C05458=1092.855,441.549,394.876,178.684,26.061,154.074
C05459=1092.862,441.795,394.832,178.687,26.074,154.077
C05460=1092.868,442.041,394.788,178.690,26.088,154.080
C05461=1092.875,442.287,394.744,178.693,26.101,154.083
C05462=1092.881,442.532,394.701,178.697,26.115,154.086
C05463=1092.888,442.778,394.656,178.700,26.128,154.089
C05464=1092.894,443.024,394.612,178.703,26.142,154.092
C05465=1092.901,443.270,394.568,178.707,26.155,154.095
C05466=1092.908,443.516,394.523,178.710,26.169,154.098
C05467=1092.914,443.762,394.479,178.713,26.182,154.101
C05468=1092.921,444.007,394.435,178.716,26.196,154.104
C05469=1092.927,444.253,394.390,178.719,26.210,154.107
C05470=1092.934,444.499,394.346,178.723,26.224,154.110
C05471=1092.941,444.745,394.302,178.725,26.237,154.114
C05472=1092.947,444.991,394.257,178.728,26.251,154.117
C05473=1092.954,445.237,394.213,178.730,26.265,154.120
C05474=1092.960,445.482,394.169,178.733,26.279,154.123
C05475=1092.968,445.728,394.124,178.735,26.292,154.126
C05476=1092.973,445.974,394.079,178.737,26.306,154.130
C05477=1092.980,446.220,394.035,178.738,26.319,154.133
C05478=1092.988,446.466,393.990,178.741,26.333,154.136
C05479=1092.994,446.712,393.946,178.741,26.347,154.140
C05480=1093.000,446.958,393.901,178.743,26.361,154.143
C05481=1093.007,447.204,393.856,178.744,26.374,154.146
C05482=1093.014,447.449,393.811,178.745,26.388,154.150
C05483=1093.020,447.695,393.767,178.746,26.401,154.153
C05484=1093.027,447.941,393.722,178.747,26.415,154.156
C05485=1093.034,448.187,393.677,178.747,26.429,154.160
C05486=1093.040,448.432,393.632,178.747,26.442,154.163
C05487=1093.047,448.678,393.587,178.748,26.456,154.166
C05488=1093.054,448.924,393.543,178.748,26.469,154.170
C05489=1093.060,449.170,393.497,178.748,26.483,154.173
C05490=1093.067,449.415,393.453,178.747,26.496,154.177
C05491=1093.074,449.661,393.408,178.748,26.510,154.180
C05492=1093.081,449.906,393.363,178.748,26.523,154.184
C05493=1093.089,450.153,393.319,178.747,26.535,154.187
C05494=1092.703,450.144,393.142,178.697,26.740,154.244
C05495=1092.694,449.897,393.187,178.697,26.727,154.241
C05496=1092.687,449.651,393.232,178.698,26.714,154.237
C05497=1092.680,449.406,393.276,178.698,26.700,154.234
C05498=1092.673,449.161,393.321,178.698,26.686,154.230
C05499=1092.667,448.915,393.366,178.698,26.673,154.227
C05500=1092.660,448.669,393.411,178.698,26.660,154.224
C05501=1092.653,448.423,393.456,178.697,26.646,154.220
C05502=1092.647,448.177,393.501,178.697,26.633,154.217
C05503=1092.640,447.932,393.546,178.697,26.619,154.213
C05504=1092.633,447.686,393.591,178.695,26.605,154.210
C05505=1092.627,447.440,393.636,178.695,26.591,154.207
C05506=1092.620,447.195,393.680,178.694,26.578,154.203
C05507=1092.613,446.949,393.725,178.692,26.564,154.200
C05508=1092.607,446.702,393.770,178.691,26.550,154.197
C05509=1092.600,446.457,393.814,178.689,26.536,154.193
C05510=1092.593,446.211,393.859,178.687,26.523,154.190
C05511=1092.586,445.966,393.904,178.686,26.509,154.187
C05512=1092.580,445.719,393.948,178.684,26.495,154.183
C05513=1092.573,445.473,393.993,178.682,26.482,154.180
C05514=1092.566,445.228,394.038,178.679,26.468,154.177
C05515=1092.560,444.982,394.082,178.677,26.454,154.174
C05516=1092.553,444.736,394.126,178.674,26.440,154.170
C05517=1092.547,444.490,394.172,178.671,26.427,154.167
C05518=1092.540,444.244,394.215,178.668,26.413,154.164
C05519=1092.533,443.999,394.260,178.664,26.399,154.161
C05520=1092.526,443.752,394.304,178.661,26.385,154.158
C05521=1092.520,443.507,394.349,178.658,26.371,154.155
C05522=1092.513,443.261,394.393,178.655,26.358,154.152
C05523=1092.507,443.016,394.437,178.651,26.344,154.149
C05524=1092.500,442.770,394.481,178.647,26.330,154.146
C05525=1092.493,442.524,394.526,178.644,26.317,154.143
C05526=1092.487,442.278,394.569,178.641,26.303,154.139
C05527=1092.480,442.032,394.614,178.638,26.290,154.136
C05528=1092.474,441.786,394.658,178.634,26.276,154.133
C05529=1092.467,441.540,394.702,178.631,26.263,154.130
C05530=1092.460,441.294,394.746,178.628,26.250,154.127
C05531=1092.454,441.048,394.790,178.624,26.237,154.125
C05532=1092.448,440.802,394.834,178.621,26.224,154.122
C05533=1092.441,440.556,394.878,178.618,26.210,154.119
C05534=1092.434,440.311,394.922,178.614,26.197,154.116
C05535=1092.428,440.065,394.966,178.611,26.185,154.113
C05536=1092.421,439.818,395.010,178.608,26.171,154.110
C05537=1092.414,439.573,395.053,178.604,26.158,154.107
C05538=1092.407,439.327,395.097,178.601,26.146,154.104
C05539=1092.397,438.921,395.169,178.596,26.124,154.099
C05540=1092.386,438.515,395.241,178.590,26.104,154.095
C05541=1092.375,438.111,395.313,178.585,26.083,154.090
C05542=1092.364,437.705,395.384,178.579,26.062,154.086
C05543=1092.358,437.459,395.428,178.576,26.050,154.083
C05544=1092.351,437.214,395.471,178.573,26.037,154.080
C05545=1092.345,436.967,395.514,178.570,26.025,154.077
C05546=1092.338,436.721,395.558,178.566,26.012,154.075
C05547=1092.331,436.475,395.602,178.562,25.999,154.072
C05548=1092.325,436.229,395.645,178.560,25.987,154.069
C05549=1092.319,435.983,395.689,178.556,25.975,154.066
C05550=1092.311,435.737,395.732,178.553,25.963,154.064
C05551=1092.306,435.491,395.775,178.550,25.951,154.061
C05552=1092.300,435.245,395.818,178.546,25.938,154.058
C05553=1092.293,434.999,395.861,178.544,25.927,154.056
C05554=1092.286,434.753,395.905,178.540,25.914,154.053
C05555=1092.279,434.507,395.947,178.537,25.902,154.050
C05556=1092.273,434.260,395.990,178.533,25.890,154.048
C05557=1092.267,434.015,396.034,178.530,25.878,154.045
C05558=1092.261,433.769,396.076,178.527,25.866,154.042
C05559=1092.254,433.522,396.120,178.524,25.854,154.040
C05560=1092.247,433.276,396.163,178.521,25.843,154.037
C05561=1092.242,433.030,396.206,178.517,25.831,154.035
C05562=1092.235,432.784,396.248,178.514,25.819,154.032
C05563=1092.229,432.538,396.291,178.510,25.807,154.029
C05564=1092.222,432.291,396.334,178.508,25.796,154.027
C05565=1092.215,432.046,396.377,178.505,25.784,154.024
C05566=1092.209,431.800,396.420,178.501,25.772,154.022
C05567=1092.202,431.553,396.462,178.498,25.761,154.019
C05568=1092.196,431.307,396.506,178.495,25.750,154.017
C05569=1092.189,431.061,396.548,178.491,25.738,154.014
C05570=1092.183,430.815,396.590,178.488,25.726,154.012
C05571=1092.177,430.568,396.633,178.485,25.716,154.010
C05572=1092.170,430.322,396.676,178.481,25.704,154.007
C05573=1092.164,430.077,396.718,178.478,25.692,154.005
C05574=1092.158,429.830,396.761,178.475,25.681,154.002
C05575=1092.151,429.584,396.804,178.472,25.670,154.000
C05576=1092.145,429.337,396.845,178.469,25.659,153.997
C05577=1092.138,429.091,396.888,178.466,25.648,153.995
C05578=1092.132,428.845,396.931,178.463,25.637,153.993
C05579=1092.126,428.599,396.973,178.459,25.625,153.990
C05580=1092.119,428.352,397.015,178.456,25.614,153.988
C05581=1092.112,428.106,397.057,178.453,25.603,153.985
C05582=1092.106,427.860,397.100,178.449,25.593,153.983
C05583=1092.100,427.613,397.141,178.447,25.582,153.981
C05584=1092.093,427.367,397.185,178.443,25.571,153.978
C05585=1092.087,427.121,397.227,178.440,25.560,153.976
C05586=1092.081,426.874,397.269,178.437,25.549,153.974
C05587=1092.074,426.629,397.311,178.433,25.539,153.972
C05588=1092.068,426.382,397.353,178.430,25.528,153.969
C05589=1092.062,426.136,397.395,178.427,25.518,153.967
C05590=1092.055,425.889,397.437,178.423,25.507,153.965
C05591=1092.049,425.658,397.476,178.421,25.497,153.963
C05592=1092.043,425.427,397.515,178.418,25.487,153.961
C05593=1092.037,425.196,397.555,178.415,25.477,153.958
C05594=1092.031,424.965,397.594,178.411,25.467,153.956
C05595=1092.025,424.733,397.634,178.409,25.457,153.954
C05596=1092.019,424.503,397.673,178.406,25.447,153.952
C05597=1092.013,424.271,397.713,178.403,25.437,153.950
C05598=1092.008,424.040,397.751,178.399,25.427,153.948
C05599=1092.001,423.793,397.794,178.396,25.417,153.946
C05600=1091.995,423.547,397.835,178.393,25.407,153.944
C05601=1091.988,423.300,397.877,178.390,25.396,153.941
C05602=1091.982,423.054,397.918,178.387,25.386,153.939
C05603=1091.976,422.807,397.960,178.384,25.376,153.937
C05604=1091.970,422.562,398.002,178.381,25.366,153.935
C05605=1091.963,422.315,398.044,178.377,25.356,153.933
C05606=1091.957,422.069,398.086,178.374,25.345,153.931
C05607=1091.951,421.822,398.127,178.371,25.335,153.929
C05608=1091.944,421.576,398.168,178.368,25.325,153.926
C05609=1091.938,421.330,398.210,178.365,25.316,153.924
C05610=1091.931,421.083,398.252,178.362,25.305,153.922
C05611=1091.925,420.836,398.293,178.358,25.295,153.920
C05612=1091.919,420.591,398.334,178.355,25.286,153.918
C05613=1091.913,420.343,398.375,178.352,25.275,153.916
C05614=1091.907,420.097,398.416,178.349,25.266,153.914
C05615=1091.900,419.850,398.458,178.345,25.256,153.912
C05616=1091.893,419.604,398.499,178.342,25.246,153.910
C05617=1091.887,419.358,398.541,178.339,25.236,153.908
C05618=1091.881,419.111,398.582,178.336,25.227,153.906
C05619=1091.874,418.864,398.623,178.334,25.217,153.904
C05620=1091.869,418.618,398.664,178.330,25.208,153.902
C05621=1091.863,418.372,398.705,178.327,25.198,153.900
C05622=1091.856,418.124,398.747,178.324,25.188,153.898
C05623=1091.850,417.879,398.787,178.321,25.179,153.896
C05624=1091.844,417.632,398.829,178.317,25.169,153.894
C05625=1091.838,417.386,398.870,178.314,25.159,153.892
C05626=1091.831,417.139,398.911,178.311,25.150,153.890
C05627=1091.821,416.758,398.974,178.306,25.135,153.887
C05628=1091.812,416.375,399.038,178.301,25.120,153.884
C05629=1091.803,415.993,399.101,178.296,25.106,153.881
C05630=1091.793,415.612,399.165,178.292,25.092,153.878
C05631=1091.786,415.365,399.205,178.288,25.082,153.876
C05632=1091.780,415.119,399.245,178.286,25.074,153.874
C05633=1091.773,414.872,399.287,178.282,25.064,153.873
C05634=1091.767,414.625,399.327,178.279,25.055,153.871
C05635=1091.761,414.378,399.368,178.276,25.046,153.869
C05636=1091.755,414.133,399.409,178.273,25.037,153.867
C05637=1091.748,413.886,399.449,178.270,25.028,153.865
C05638=1091.742,413.638,399.490,178.267,25.018,153.863
C05639=1091.736,413.392,399.530,178.263,25.010,153.861
C05640=1091.730,413.146,399.571,178.261,25.001,153.860
C05641=1091.723,412.899,399.612,178.258,24.992,153.858
C05642=1091.717,412.653,399.652,178.254,24.983,153.856
C05643=1091.711,412.406,399.692,178.251,24.973,153.854
C05644=1091.705,412.159,399.733,178.248,24.965,153.852
C05645=1091.698,411.913,399.773,178.245,24.956,153.851
C05646=1091.692,411.665,399.814,178.242,24.947,153.849
C05647=1091.685,411.354,399.865,178.238,24.936,153.847
C05648=1091.676,411.041,399.916,178.234,24.925,153.844
C05649=1091.668,410.729,399.967,178.230,24.914,153.842
C05650=1091.661,410.417,400.017,178.226,24.903,153.840
C05651=1091.655,410.170,400.058,178.223,24.894,153.838
C05652=1091.649,409.924,400.098,178.221,24.885,153.836
C05653=1091.642,409.677,400.138,178.217,24.877,153.835
C05654=1091.636,409.431,400.179,178.214,24.868,153.833
C05655=1091.631,409.183,400.219,178.211,24.860,153.831
C05656=1091.624,408.937,400.259,178.208,24.851,153.829
C05657=1091.618,408.690,400.299,178.205,24.842,153.828
C05658=1091.611,408.444,400.339,178.202,24.834,153.826
C05659=1091.606,408.196,400.379,178.198,24.825,153.824
C05660=1091.600,407.950,400.419,178.196,24.817,153.823
C05661=1091.593,407.703,400.459,178.192,24.808,153.821
C05662=1091.587,407.457,400.500,178.190,24.800,153.819
C05663=1091.581,407.210,400.539,178.186,24.791,153.818
C05664=1091.575,406.963,400.579,178.184,24.783,153.816
C05665=1091.568,406.716,400.619,178.180,24.775,153.814
C05666=1091.562,406.469,400.659,178.177,24.767,153.813
C05667=1091.557,406.223,400.699,178.174,24.758,153.811
C05668=1091.551,405.976,400.739,178.171,24.750,153.809
C05669=1091.545,405.730,400.779,178.168,24.742,153.808
C05670=1091.539,405.482,400.818,178.165,24.734,153.806
C05671=1091.532,405.236,400.858,178.162,24.725,153.805
C05672=1091.526,404.989,400.898,178.159,24.718,153.803
C05673=1091.520,404.742,400.937,178.156,24.709,153.801
C05674=1091.514,404.495,400.977,178.153,24.701,153.800
C05675=1091.508,404.249,401.016,178.149,24.693,153.798
C05676=1091.501,404.003,401.056,178.147,24.685,153.797
C05677=1091.495,403.755,401.095,178.143,24.677,153.795
C05678=1091.489,403.508,401.135,178.141,24.669,153.794
C05679=1091.483,403.261,401.174,178.138,24.661,153.792
C05680=1091.476,403.015,401.214,178.134,24.653,153.791
C05681=1091.471,402.768,401.253,178.132,24.645,153.789
C05682=1091.465,402.521,401.293,178.128,24.637,153.787
C05683=1091.458,402.274,401.332,178.125,24.630,153.786
C05684=1091.452,402.028,401.372,178.123,24.622,153.784
C05685=1091.446,401.781,401.411,178.119,24.614,153.783
C05686=1091.440,401.534,401.450,178.116,24.606,153.781
C05687=1091.434,401.287,401.490,178.113,24.598,153.780
C05688=1091.427,401.040,401.529,178.110,24.591,153.778
C05689=1091.422,400.794,401.568,178.107,24.583,153.777
C05690=1091.416,400.547,401.607,178.104,24.575,153.775
C05691=1091.410,400.299,401.647,178.101,24.568,153.774
C05692=1091.403,400.053,401.685,178.098,24.560,153.772
C05693=1091.397,399.806,401.724,178.095,24.552,153.771
C05694=1091.391,399.559,401.764,178.092,24.544,153.769
C05695=1091.385,399.312,401.803,178.089,24.537,153.768
C05696=1091.379,399.066,401.842,178.086,24.529,153.767
C05697=1091.373,398.819,401.881,178.083,24.522,153.765
C05698=1091.367,398.572,401.921,178.080,24.514,153.764
C05699=1091.361,398.349,401.956,178.077,24.508,153.762
C05700=1091.355,398.126,401.991,178.074,24.500,153.761
C05701=1091.351,397.902,402.026,178.071,24.494,153.760
C05702=1091.345,397.679,402.061,178.069,24.487,153.759
C05703=1091.339,397.455,402.097,178.066,24.480,153.757
C05704=1091.333,397.232,402.132,178.063,24.474,153.756
C05705=1091.328,397.008,402.166,178.060,24.467,153.755
C05706=1091.323,396.785,402.202,178.058,24.461,153.753
C05707=1091.316,396.538,402.241,178.055,24.453,153.752
C05708=1091.311,396.291,402.279,178.052,24.446,153.751
C05709=1091.304,396.044,402.318,178.049,24.438,153.749
C05710=1091.299,395.798,402.357,178.046,24.431,153.748
C05711=1091.292,395.551,402.395,178.043,24.424,153.747
C05712=1091.287,395.304,402.434,178.040,24.417,153.745
C05713=1091.280,395.057,402.473,178.037,24.409,153.744
C05714=1091.275,394.810,402.512,178.034,24.402,153.742
C05715=1091.268,394.563,402.550,178.030,24.395,153.741
C05716=1091.262,394.316,402.589,178.028,24.388,153.740
C05717=1091.256,394.070,402.628,178.025,24.380,153.738
C05718=1091.249,393.823,402.666,178.022,24.373,153.737
C05719=1091.244,393.576,402.705,178.019,24.367,153.736
C05720=1091.237,393.328,402.743,178.015,24.359,153.734
C05721=1091.232,393.082,402.782,178.012,24.352,153.733
C05722=1091.226,392.835,402.820,178.009,24.345,153.732
C05723=1091.219,392.588,402.859,178.007,24.338,153.730
C05724=1091.214,392.341,402.897,178.004,24.331,153.729
C05725=1091.207,392.094,402.936,178.001,24.324,153.728
C05726=1091.201,391.848,402.974,177.997,24.317,153.727
C05727=1091.195,391.600,403.012,177.994,24.310,153.725
C05728=1091.189,391.354,403.051,177.991,24.303,153.724
C05729=1091.183,391.106,403.089,177.988,24.296,153.723
C05730=1091.177,390.860,403.127,177.985,24.290,153.722
C05731=1091.171,390.613,403.165,177.982,24.283,153.720
C05732=1091.164,390.366,403.203,177.979,24.275,153.719
C05733=1091.158,390.119,403.241,177.976,24.269,153.718
C05734=1091.152,389.872,403.279,177.973,24.262,153.717
C05735=1091.147,389.625,403.317,177.970,24.255,153.715
C05736=1091.140,389.379,403.356,177.967,24.249,153.714
C05737=1091.134,389.131,403.394,177.964,24.242,153.713
C05738=1091.128,388.884,403.432,177.961,24.235,153.712
C05739=1091.122,388.638,403.470,177.957,24.228,153.710
C05740=1091.116,388.390,403.508,177.954,24.222,153.709
C05741=1091.110,388.143,403.545,177.951,24.215,153.708
C05742=1091.104,387.897,403.583,177.948,24.208,153.707
C05743=1091.098,387.650,403.621,177.945,24.202,153.706
C05744=1091.091,387.403,403.659,177.943,24.195,153.704
C05745=1091.086,387.156,403.697,177.939,24.189,153.703
C05746=1091.080,386.909,403.735,177.937,24.182,153.702
C05747=1091.074,386.662,403.773,177.934,24.175,153.701
C05748=1091.068,386.415,403.811,177.931,24.169,153.700
C05749=1091.062,386.168,403.849,177.927,24.162,153.699
C05750=1091.056,385.921,403.887,177.924,24.156,153.697
C05751=1091.050,385.674,403.924,177.921,24.149,153.696
C05752=1091.044,385.427,403.962,177.918,24.143,153.695
C05753=1091.038,385.180,404.000,177.915,24.136,153.694
C05754=1091.032,384.933,404.038,177.912,24.130,153.693
C05755=1091.026,384.716,404.071,177.910,24.124,153.692
C05756=1091.021,384.500,404.103,177.906,24.118,153.691
C05757=1091.016,384.282,404.137,177.904,24.113,153.690
C05758=1091.011,384.066,404.169,177.901,24.107,153.689
C05759=1091.005,383.849,404.203,177.898,24.101,153.688
C05760=1091.000,383.633,404.236,177.896,24.095,153.687
C05761=1090.995,383.416,404.269,177.893,24.090,153.686
C05762=1090.991,383.199,404.302,177.891,24.084,153.685
C05763=1090.985,382.952,404.339,177.888,24.078,153.684
C05764=1090.978,382.705,404.376,177.885,24.072,153.682
C05765=1090.972,382.458,404.414,177.882,24.065,153.681
C05766=1090.966,382.211,404.452,177.879,24.059,153.680
C05767=1090.960,381.964,404.489,177.875,24.053,153.679
C05768=1090.954,381.717,404.527,177.872,24.047,153.678
C05769=1090.948,381.470,404.563,177.869,24.040,153.677
C05770=1090.942,381.223,404.601,177.866,24.034,153.676
C05771=1090.937,380.976,404.638,177.863,24.028,153.675
C05772=1090.930,380.729,404.675,177.860,24.022,153.674
C05773=1090.924,380.481,404.712,177.857,24.016,153.673
C05774=1090.918,380.234,404.750,177.854,24.010,153.672
C05775=1090.912,379.987,404.787,177.851,24.003,153.671
C05776=1090.906,379.741,404.824,177.848,23.997,153.670
C05777=1090.900,379.493,404.861,177.845,23.991,153.669
C05778=1090.894,379.246,404.898,177.842,23.985,153.667
C05779=1090.888,378.999,404.936,177.839,23.979,153.666
C05780=1090.882,378.752,404.973,177.835,23.973,153.665
C05781=1090.877,378.505,405.010,177.832,23.967,153.664
C05782=1090.870,378.258,405.047,177.829,23.961,153.663
C05783=1090.864,378.011,405.084,177.827,23.955,153.662
C05784=1090.859,377.764,405.121,177.824,23.949,153.661
C05785=1090.852,377.517,405.157,177.821,23.943,153.660
C05786=1090.846,377.270,405.195,177.818,23.937,153.659
C05787=1090.840,377.023,405.231,177.814,23.931,153.658
C05788=1090.835,376.775,405.269,177.811,23.925,153.657
C05789=1090.829,376.528,405.306,177.808,23.919,153.656
C05790=1090.823,376.281,405.342,177.805,23.913,153.655
C05791=1090.817,376.034,405.380,177.802,23.907,153.654
C05792=1090.811,375.787,405.417,177.799,23.901,153.653
C05793=1090.805,375.540,405.453,177.796,23.895,153.652
C05794=1090.799,375.292,405.490,177.793,23.890,153.651
C05795=1090.793,375.045,405.527,177.790,23.884,153.650
C05796=1090.787,374.798,405.564,177.787,23.878,153.649
C05797=1090.781,374.551,405.600,177.784,23.872,153.648
C05798=1090.775,374.304,405.637,177.781,23.866,153.647
C05799=1090.769,374.057,405.674,177.778,23.860,153.646
C05800=1090.763,373.809,405.711,177.774,23.855,153.645
C05801=1090.758,373.563,405.747,177.771,23.849,153.644
C05802=1090.752,373.315,405.784,177.769,23.843,153.643
C05803=1090.746,373.068,405.820,177.766,23.837,153.642
C05804=1090.740,372.821,405.856,177.763,23.832,153.641
C05805=1090.734,372.573,405.893,177.759,23.826,153.641
C05806=1090.728,372.326,405.930,177.756,23.820,153.640
C05807=1090.721,372.079,405.966,177.753,23.814,153.639
C05808=1090.716,371.832,406.003,177.750,23.809,153.638
C05809=1090.710,371.584,406.039,177.747,23.804,153.637
C05810=1090.703,371.337,406.075,177.744,23.798,153.636
C05811=1090.694,370.932,406.135,177.739,23.789,153.634
C05812=1090.684,370.525,406.195,177.734,23.779,153.633
C05813=1090.675,370.119,406.255,177.729,23.770,153.631
C05814=1090.665,369.714,406.314,177.724,23.761,153.630
C05815=1090.659,369.467,406.350,177.721,23.756,153.629
C05816=1090.652,369.220,406.387,177.718,23.750,153.628
C05817=1090.647,368.972,406.423,177.715,23.744,153.627
C05818=1090.641,368.725,406.459,177.712,23.739,153.626
C05819=1090.635,368.478,406.495,177.708,23.734,153.626
C05820=1090.629,368.231,406.531,177.706,23.728,153.625
C05821=1090.624,367.983,406.568,177.703,23.723,153.624
C05822=1090.618,367.736,406.604,177.699,23.717,153.623
C05823=1090.612,367.489,406.639,177.696,23.712,153.622
C05824=1090.605,367.242,406.676,177.693,23.706,153.621
C05825=1090.600,366.994,406.712,177.691,23.701,153.620
C05826=1090.594,366.747,406.748,177.687,23.696,153.619
C05827=1090.588,366.500,406.784,177.684,23.690,153.618
C05828=1090.582,366.252,406.820,177.681,23.684,153.618
C05829=1090.577,366.006,406.856,177.678,23.679,153.617
C05830=1090.571,365.758,406.892,177.675,23.674,153.616
C05831=1090.565,365.510,406.928,177.672,23.669,153.615
C05832=1090.559,365.263,406.964,177.668,23.663,153.614
C05833=1090.553,365.016,407.000,177.666,23.658,153.613
C05834=1090.547,364.768,407.035,177.663,23.653,153.613
C05835=1090.541,364.521,407.071,177.659,23.647,153.612
C05836=1090.535,364.273,407.108,177.657,23.642,153.611
C05837=1090.530,364.027,407.143,177.654,23.637,153.610
C05838=1090.524,363.779,407.179,177.650,23.632,153.609
C05839=1090.518,363.531,407.214,177.647,23.627,153.609
C05840=1090.512,363.284,407.250,177.645,23.622,153.608
C05841=1090.506,363.037,407.286,177.641,23.616,153.607
C05842=1090.500,362.789,407.322,177.638,23.611,153.606
C05843=1090.494,362.543,407.357,177.636,23.606,153.605
C05844=1090.488,362.295,407.392,177.632,23.601,153.604
C05845=1090.482,362.047,407.428,177.629,23.595,153.604
C05846=1090.476,361.800,407.464,177.625,23.590,153.603
C05847=1090.470,361.553,407.499,177.623,23.585,153.602
C05848=1090.464,361.305,407.535,177.620,23.580,153.601
C05849=1090.459,361.058,407.570,177.616,23.575,153.601
C05850=1090.453,360.810,407.606,177.614,23.570,153.600
C05851=1090.447,360.563,407.641,177.611,23.565,153.599
C05852=1090.441,360.316,407.677,177.607,23.560,153.598
C05853=1090.434,360.068,407.712,177.605,23.555,153.597
C05854=1090.429,359.821,407.748,177.601,23.550,153.597
C05855=1090.423,359.574,407.783,177.598,23.545,153.596
C05856=1090.418,359.327,407.819,177.596,23.540,153.595
C05857=1090.412,359.079,407.854,177.592,23.535,153.594
C05858=1090.405,358.831,407.889,177.589,23.530,153.594
C05859=1090.400,358.584,407.924,177.586,23.525,153.593
C05860=1090.394,358.337,407.960,177.583,23.520,153.592
C05861=1090.388,358.090,407.995,177.579,23.515,153.591
C05862=1090.381,357.842,408.031,177.577,23.510,153.591
C05863=1090.373,357.451,408.086,177.571,23.502,153.590
C05864=1090.363,357.062,408.141,177.567,23.494,153.588
C05865=1090.355,356.671,408.197,177.562,23.486,153.587
C05866=1090.345,356.280,408.252,177.558,23.479,153.586
C05867=1090.340,356.033,408.287,177.554,23.474,153.585
C05868=1090.333,355.785,408.322,177.551,23.469,153.585
C05869=1090.327,355.538,408.358,177.548,23.464,153.584
C05870=1090.322,355.290,408.393,177.545,23.459,153.583
C05871=1090.315,355.043,408.427,177.542,23.454,153.582
C05872=1090.310,354.795,408.462,177.539,23.449,153.582
C05873=1090.304,354.548,408.498,177.536,23.444,153.581
C05874=1090.298,354.300,408.532,177.533,23.440,153.580
C05875=1090.292,354.053,408.568,177.530,23.435,153.580
C05876=1090.286,353.805,408.602,177.527,23.430,153.579
C05877=1090.281,353.558,408.637,177.524,23.425,153.578
C05878=1090.275,353.310,408.672,177.520,23.420,153.577
C05879=1090.269,353.063,408.707,177.518,23.416,153.577
C05880=1090.263,352.816,408.742,177.514,23.411,153.576
C05881=1090.257,352.568,408.777,177.512,23.407,153.575
C05882=1090.252,352.321,408.812,177.508,23.402,153.575
C05883=1090.245,352.073,408.846,177.505,23.397,153.574
C05884=1090.240,351.826,408.881,177.502,23.392,153.573
C05885=1090.233,351.578,408.916,177.499,23.387,153.573
C05886=1090.227,351.331,408.950,177.496,23.383,153.572
C05887=1090.222,351.084,408.985,177.493,23.378,153.571
C05888=1090.216,350.836,409.020,177.490,23.374,153.571
C05889=1090.210,350.588,409.054,177.487,23.369,153.570
C05890=1090.204,350.340,409.089,177.484,23.364,153.569
C05891=1090.198,350.093,409.124,177.481,23.360,153.569
C05892=1090.193,349.846,409.158,177.477,23.355,153.568
C05893=1090.186,349.598,409.192,177.475,23.350,153.567
C05894=1090.181,349.350,409.227,177.471,23.346,153.567
C05895=1090.175,349.103,409.261,177.469,23.341,153.566
C05896=1090.169,348.855,409.296,177.465,23.337,153.566
C05897=1090.164,348.607,409.330,177.462,23.332,153.565
C05898=1090.157,348.361,409.365,177.459,23.327,153.564
C05899=1090.152,348.112,409.400,177.456,23.323,153.564
C05900=1090.146,347.865,409.434,177.453,23.318,153.563
C05901=1090.140,347.618,409.468,177.450,23.314,153.562
C05902=1090.135,347.370,409.503,177.447,23.309,153.562
C05903=1090.128,347.122,409.537,177.444,23.305,153.561
C05904=1090.123,346.875,409.571,177.441,23.300,153.560
C05905=1090.117,346.628,409.605,177.438,23.296,153.560
C05906=1090.111,346.379,409.640,177.434,23.291,153.559
C05907=1090.105,346.132,409.674,177.432,23.287,153.559
C05908=1090.099,345.885,409.708,177.428,23.282,153.558
C05909=1090.094,345.637,409.743,177.426,23.278,153.557
C05910=1090.088,345.389,409.777,177.422,23.273,153.557
C05911=1090.082,345.141,409.811,177.420,23.269,153.556
C05912=1090.076,344.894,409.845,177.416,23.264,153.555
C05913=1090.070,344.647,409.879,177.413,23.260,153.555
C05914=1090.065,344.398,409.914,177.410,23.255,153.554
C05915=1090.055,344.010,409.967,177.405,23.248,153.553
C05916=1090.046,343.623,410.020,177.400,23.241,153.552
C05917=1090.037,343.235,410.074,177.395,23.234,153.551
C05918=1090.028,342.847,410.126,177.391,23.228,153.551
C05919=1090.022,342.600,410.160,177.388,23.223,153.550
C05920=1090.016,342.353,410.195,177.384,23.219,153.549
C05921=1090.011,342.105,410.228,177.382,23.215,153.549
C05922=1090.004,341.857,410.262,177.379,23.211,153.548
C05923=1089.998,341.610,410.296,177.375,23.206,153.548
C05924=1089.993,341.362,410.330,177.373,23.202,153.547
C05925=1089.987,341.114,410.364,177.369,23.197,153.547
C05926=1089.981,340.866,410.397,177.366,23.193,153.546
C05927=1089.975,340.619,410.431,177.363,23.189,153.545
C05928=1089.970,340.372,410.465,177.360,23.185,153.545
C05929=1089.963,340.123,410.499,177.357,23.180,153.544
C05930=1089.958,339.876,410.533,177.354,23.176,153.544
C05931=1089.952,339.628,410.566,177.351,23.172,153.543
C05932=1089.946,339.381,410.600,177.348,23.167,153.543
C05933=1089.941,339.133,410.634,177.345,23.163,153.542
C05934=1089.935,338.886,410.668,177.342,23.159,153.541
C05935=1089.929,338.638,410.701,177.339,23.155,153.541
C05936=1089.924,338.390,410.734,177.336,23.151,153.540
C05937=1089.918,338.142,410.768,177.332,23.146,153.540
C05938=1089.912,337.895,410.802,177.330,23.142,153.539
C05939=1089.906,337.647,410.836,177.326,23.138,153.539
C05940=1089.900,337.399,410.870,177.323,23.134,153.538
C05941=1089.894,337.151,410.902,177.321,23.130,153.538
C05942=1089.888,336.904,410.936,177.317,23.125,153.537
C05943=1089.882,336.656,410.970,177.314,23.122,153.537
C05944=1089.877,336.408,411.003,177.311,23.117,153.536
C05945=1089.871,336.160,411.036,177.308,23.113,153.535
C05946=1089.865,335.913,411.070,177.305,23.109,153.535
C05947=1089.859,335.665,411.103,177.302,23.105,153.534
C05948=1089.854,335.417,411.136,177.299,23.101,153.534
C05949=1089.848,335.169,411.170,177.296,23.097,153.533
C05950=1089.842,334.922,411.204,177.293,23.092,153.533
C05951=1089.836,334.675,411.237,177.290,23.088,153.532
C05952=1089.830,334.427,411.270,177.287,23.085,153.532
C05953=1089.825,334.179,411.303,177.284,23.080,153.531
C05954=1089.819,333.931,411.337,177.281,23.076,153.531
C05955=1089.813,333.683,411.369,177.277,23.072,153.530
C05956=1089.807,333.435,411.403,177.275,23.068,153.530
C05957=1089.802,333.187,411.436,177.272,23.064,153.529
C05958=1089.795,332.940,411.470,177.268,23.059,153.529
C05959=1089.790,332.693,411.503,177.265,23.056,153.528
C05960=1089.784,332.445,411.536,177.263,23.052,153.528
C05961=1089.779,332.197,411.570,177.259,23.047,153.527
C05962=1089.772,331.949,411.602,177.256,23.043,153.527
C05963=1089.767,331.701,411.636,177.253,23.040,153.526
C05964=1089.761,331.454,411.668,177.250,23.036,153.526
C05965=1089.755,331.206,411.702,177.247,23.032,153.525
C05966=1089.749,330.958,411.734,177.244,23.028,153.525
C05967=1089.740,330.564,411.787,177.239,23.022,153.524
C05968=1089.730,330.170,411.839,177.234,23.015,153.523
C05969=1089.720,329.777,411.890,177.229,23.009,153.523
C05970=1089.711,329.383,411.944,177.224,23.003,153.522
C05971=1089.706,329.136,411.975,177.221,22.999,153.521
C05972=1089.700,328.888,412.009,177.219,22.995,153.521
C05973=1089.694,328.640,412.041,177.216,22.992,153.521
C05974=1089.688,328.392,412.075,177.212,22.987,153.520
C05975=1089.682,328.145,412.107,177.209,22.984,153.520
C05976=1089.676,327.897,412.139,177.206,22.980,153.519
C05977=1089.671,327.649,412.173,177.203,22.976,153.519
C05978=1089.664,327.401,412.206,177.200,22.972,153.518
C05979=1089.658,327.153,412.238,177.197,22.968,153.518
C05980=1089.653,326.906,412.271,177.194,22.965,153.517
C05981=1089.647,326.658,412.303,177.191,22.960,153.517
C05982=1089.642,326.410,412.336,177.188,22.957,153.516
C05983=1089.636,326.162,412.369,177.185,22.953,153.516
C05984=1089.629,325.914,412.401,177.182,22.949,153.516
C05985=1089.624,325.666,412.434,177.178,22.945,153.515
C05986=1089.618,325.419,412.466,177.176,22.942,153.515
C05987=1089.612,325.171,412.498,177.173,22.938,153.514
C05988=1089.606,324.923,412.531,177.170,22.934,153.514
C05989=1089.601,324.675,412.564,177.166,22.930,153.513
C05990=1089.594,324.427,412.597,177.163,22.926,153.513
C05991=1089.589,324.180,412.629,177.161,22.923,153.513
C05992=1089.584,323.932,412.662,177.158,22.919,153.512
C05993=1089.578,323.683,412.694,177.154,22.914,153.512
C05994=1089.571,323.436,412.726,177.151,22.911,153.511
C05995=1089.567,323.188,412.759,177.149,22.908,153.511
C05996=1089.560,322.940,412.791,177.146,22.904,153.510
C05997=1089.554,322.692,412.823,177.142,22.900,153.510
C05998=1089.549,322.445,412.856,177.139,22.896,153.510
C05999=1089.543,322.197,412.888,177.136,22.892,153.509
C06000=1089.537,321.949,412.920,177.134,22.889,153.509
C06001=1089.531,321.701,412.953,177.131,22.885,153.508
C06002=1089.526,321.453,412.985,177.127,22.881,153.508
C06003=1089.520,321.205,413.017,177.124,22.877,153.507
C06004=1089.514,320.957,413.050,177.121,22.874,153.507
C06005=1089.509,320.710,413.082,177.119,22.870,153.506
C06006=1089.503,320.462,413.114,177.116,22.866,153.506
C06007=1089.497,320.215,413.146,177.112,22.862,153.506
C06008=1089.492,319.966,413.179,177.109,22.858,153.505
C06009=1089.486,319.718,413.211,177.106,22.855,153.505
C06010=1089.481,319.470,413.242,177.103,22.852,153.504
C06011=1089.475,319.222,413.275,177.101,22.848,153.504
C06012=1089.469,318.975,413.307,177.097,22.844,153.504
C06013=1089.463,318.727,413.339,177.094,22.840,153.503
C06014=1089.458,318.479,413.372,177.091,22.836,153.503
C06015=1089.452,318.231,413.403,177.088,22.833,153.502
C06016=1089.446,317.983,413.435,177.085,22.829,153.502
C06017=1089.441,317.735,413.467,177.082,22.825,153.502
C06018=1089.435,317.487,413.499,177.079,22.822,153.501
C06019=1089.426,317.087,413.551,177.074,22.816,153.500
C06020=1089.417,316.686,413.602,177.070,22.810,153.500
C06021=1089.408,316.286,413.655,177.065,22.804,153.499
C06022=1089.398,315.885,413.706,177.060,22.798,153.498
C06023=1089.393,315.638,413.738,177.057,22.794,153.498
C06024=1089.388,315.390,413.769,177.054,22.791,153.498
C06025=1089.382,315.142,413.801,177.051,22.787,153.497
C06026=1089.376,314.894,413.833,177.048,22.783,153.497
C06027=1089.370,314.646,413.865,177.044,22.780,153.497
C06028=1089.364,314.398,413.897,177.041,22.776,153.496
C06029=1089.358,314.151,413.928,177.039,22.773,153.496
C06030=1089.352,313.902,413.959,177.036,22.770,153.495
C06031=1089.347,313.654,413.991,177.033,22.766,153.495
C06032=1089.341,313.406,414.023,177.030,22.763,153.495
C06033=1089.334,313.158,414.054,177.027,22.759,153.494
C06034=1089.329,312.911,414.086,177.023,22.755,153.494
C06035=1089.323,312.663,414.118,177.020,22.752,153.494
C06036=1089.317,312.415,414.148,177.017,22.748,153.493
C06037=1089.311,312.167,414.180,177.014,22.745,153.493
C06038=1089.306,311.919,414.212,177.012,22.741,153.493
C06039=1089.300,311.671,414.244,177.009,22.738,153.492
C06040=1089.294,311.423,414.275,177.006,22.735,153.492
C06041=1089.288,311.175,414.307,177.003,22.731,153.491
C06042=1089.283,310.927,414.338,176.999,22.728,153.491
C06043=1089.276,310.679,414.369,176.996,22.724,153.491
C06044=1089.271,310.431,414.401,176.993,22.721,153.490
C06045=1089.265,310.184,414.432,176.990,22.717,153.490
C06046=1089.259,309.935,414.463,176.987,22.714,153.490
C06047=1089.254,309.688,414.495,176.984,22.711,153.489
C06048=1089.247,309.440,414.526,176.981,22.707,153.489
C06049=1089.242,309.192,414.557,176.978,22.704,153.489
C06050=1089.236,308.943,414.589,176.976,22.700,153.488
C06051=1089.230,308.696,414.619,176.972,22.697,153.488
C06052=1089.225,308.448,414.651,176.969,22.693,153.488
C06053=1089.219,308.200,414.683,176.966,22.690,153.487
C06054=1089.213,307.952,414.713,176.963,22.687,153.487
C06055=1089.207,307.705,414.745,176.960,22.683,153.487
C06056=1089.201,307.456,414.776,176.957,22.680,153.486
C06057=1089.196,307.209,414.807,176.954,22.676,153.486
C06058=1089.190,306.961,414.838,176.951,22.673,153.486
C06059=1089.184,306.712,414.869,176.948,22.670,153.485
C06060=1089.179,306.464,414.901,176.945,22.666,153.485
C06061=1089.173,306.217,414.931,176.942,22.663,153.485
C06062=1089.167,305.968,414.963,176.939,22.659,153.484
C06063=1089.161,305.720,414.994,176.936,22.656,153.484
C06064=1089.156,305.473,415.025,176.933,22.652,153.484
C06065=1089.149,305.224,415.056,176.930,22.649,153.483
C06066=1089.144,304.976,415.087,176.927,22.646,153.483
C06067=1089.138,304.729,415.118,176.924,22.643,153.483
C06068=1089.133,304.481,415.149,176.921,22.639,153.482
C06069=1089.127,304.232,415.180,176.918,22.636,153.482
C06070=1089.121,303.985,415.211,176.915,22.633,153.482
C06071=1089.112,303.587,415.260,176.910,22.627,153.481
C06072=1089.104,303.189,415.310,176.906,22.622,153.481
C06073=1089.094,302.791,415.359,176.901,22.616,153.480
C06074=1089.085,302.394,415.409,176.895,22.610,153.480
C06075=1089.080,302.145,415.440,176.892,22.607,153.479
C06076=1089.074,301.898,415.470,176.889,22.604,153.479
C06077=1089.068,301.650,415.502,176.886,22.601,153.479
C06078=1089.063,301.402,415.532,176.884,22.597,153.478
C06079=1089.058,301.154,415.563,176.881,22.594,153.478
C06080=1089.051,300.906,415.594,176.878,22.590,153.478
C06081=1089.045,300.658,415.624,176.875,22.587,153.477
C06082=1089.040,300.410,415.655,176.872,22.584,153.477
C06083=1089.034,300.162,415.685,176.869,22.581,153.477
C06084=1089.029,299.914,415.716,176.866,22.577,153.476
C06085=1089.024,299.666,415.747,176.863,22.574,153.476
C06086=1089.018,299.418,415.778,176.860,22.571,153.476
C06087=1089.013,299.170,415.808,176.857,22.567,153.475
C06088=1089.007,298.922,415.838,176.854,22.564,153.475
C06089=1089.001,298.673,415.870,176.851,22.561,153.475
C06090=1088.995,298.425,415.900,176.848,22.557,153.474
C06091=1088.990,298.178,415.930,176.845,22.554,153.474
C06092=1088.984,297.929,415.961,176.842,22.551,153.474
C06093=1088.979,297.682,415.992,176.839,22.547,153.474
C06094=1088.973,297.434,416.022,176.836,22.544,153.473
C06095=1088.967,297.186,416.052,176.834,22.541,153.473
C06096=1088.962,296.938,416.083,176.831,22.538,153.473
C06097=1088.956,296.689,416.113,176.827,22.535,153.472
C06098=1088.950,296.441,416.144,176.824,22.532,153.472
C06099=1088.944,296.193,416.174,176.821,22.528,153.472
C06100=1088.938,295.945,416.204,176.818,22.525,153.472
C06101=1088.933,295.697,416.235,176.816,22.522,153.471
C06102=1088.927,295.449,416.264,176.813,22.519,153.471
C06103=1088.921,295.201,416.295,176.810,22.515,153.471
C06104=1088.916,294.953,416.326,176.807,22.512,153.470
C06105=1088.910,294.705,416.356,176.804,22.509,153.470
C06106=1088.905,294.457,416.386,176.801,22.506,153.470
C06107=1088.899,294.209,416.416,176.798,22.502,153.470
C06108=1088.893,293.961,416.446,176.795,22.500,153.469
C06109=1088.888,293.713,416.476,176.792,22.496,153.469
C06110=1088.882,293.465,416.506,176.789,22.493,153.469
C06111=1088.876,293.217,416.537,176.786,22.490,153.468
C06112=1088.870,292.968,416.567,176.783,22.487,153.468
C06113=1088.864,292.720,416.597,176.780,22.483,153.468
C06114=1088.858,292.472,416.627,176.777,22.480,153.468
C06115=1088.853,292.224,416.657,176.774,22.477,153.467
C06116=1088.847,291.976,416.687,176.771,22.474,153.467
C06117=1088.841,291.728,416.717,176.768,22.471,153.467
C06118=1088.836,291.480,416.747,176.765,22.468,153.467
C06119=1088.830,291.231,416.777,176.762,22.464,153.466
C06120=1088.824,290.984,416.807,176.759,22.462,153.466
C06121=1088.819,290.735,416.837,176.756,22.458,153.466
C06122=1088.814,290.488,416.867,176.753,22.455,153.465
C06123=1088.804,290.104,416.913,176.748,22.450,153.465
C06124=1088.796,289.720,416.959,176.744,22.445,153.465
C06125=1088.787,289.337,417.005,176.739,22.441,153.464
C06126=1088.777,288.953,417.052,176.735,22.436,153.464
C06127=1088.772,288.704,417.081,176.732,22.433,153.464
C06128=1088.766,288.456,417.111,176.729,22.430,153.463
C06129=1088.760,288.208,417.141,176.726,22.427,153.463
C06130=1088.754,287.960,417.170,176.723,22.424,153.463
C06131=1088.749,287.712,417.200,176.720,22.421,153.463
C06132=1088.743,287.464,417.230,176.717,22.418,153.462
C06133=1088.738,287.216,417.260,176.714,22.414,153.462
C06134=1088.732,286.968,417.289,176.711,22.412,153.462
C06135=1088.726,286.720,417.319,176.708,22.408,153.462
C06136=1088.721,286.472,417.349,176.705,22.405,153.461
C06137=1088.715,286.223,417.378,176.702,22.402,153.461
C06138=1088.709,285.975,417.407,176.699,22.399,153.461
C06139=1088.703,285.727,417.437,176.696,22.396,153.461
C06140=1088.698,285.479,417.467,176.693,22.393,153.460
C06141=1088.692,285.230,417.497,176.690,22.390,153.460
C06142=1088.686,284.983,417.526,176.688,22.387,153.460
C06143=1088.681,284.734,417.555,176.684,22.384,153.460
C06144=1088.675,284.486,417.585,176.681,22.381,153.459
C06145=1088.669,284.238,417.614,176.678,22.378,153.459
C06146=1088.664,283.989,417.644,176.675,22.375,153.459
C06147=1088.658,283.742,417.674,176.672,22.372,153.459
C06148=1088.651,283.493,417.703,176.669,22.368,153.458
C06149=1088.647,283.246,417.732,176.666,22.366,153.458
C06150=1088.641,282.997,417.762,176.663,22.362,153.458
C06151=1088.636,282.749,417.792,176.661,22.359,153.458
C06152=1088.629,282.501,417.821,176.658,22.357,153.457
C06153=1088.624,282.252,417.850,176.655,22.353,153.457
C06154=1088.618,282.005,417.879,176.652,22.351,153.457
C06155=1088.613,281.756,417.909,176.649,22.347,153.457
C06156=1088.607,281.508,417.938,176.646,22.344,153.456
C06157=1088.601,281.260,417.967,176.643,22.341,153.456
C06158=1088.596,281.012,417.996,176.640,22.338,153.456
C06159=1088.590,280.763,418.025,176.637,22.335,153.456
C06160=1088.585,280.515,418.054,176.635,22.332,153.455
C06161=1088.578,280.267,418.083,176.632,22.330,153.455
C06162=1088.573,280.018,418.113,176.629,22.326,153.455
C06163=1088.567,279.771,418.142,176.626,22.324,153.455
C06164=1088.562,279.522,418.171,176.623,22.320,153.455
C06165=1088.555,279.274,418.200,176.620,22.317,153.454
C06166=1088.550,279.025,418.229,176.617,22.314,153.454
C06167=1088.544,278.778,418.258,176.614,22.311,153.454
C06168=1088.539,278.529,418.288,176.611,22.309,153.454
C06169=1088.533,278.281,418.317,176.608,22.305,153.453
C06170=1088.527,278.033,418.346,176.605,22.303,153.453
C06171=1088.522,277.785,418.374,176.602,22.299,153.453
C06172=1088.516,277.536,418.404,176.599,22.297,153.453
C06173=1088.510,277.288,418.433,176.596,22.293,153.452
C06174=1088.506,277.040,418.462,176.593,22.291,153.452
C06175=1088.496,276.665,418.505,176.590,22.286,153.452
C06176=1088.488,276.291,418.548,176.585,22.282,153.452
C06177=1088.479,275.917,418.592,176.580,22.278,153.451
C06178=1088.470,275.543,418.635,176.576,22.273,153.451
C06179=1088.465,275.295,418.665,176.573,22.270,153.451
C06180=1088.459,275.047,418.694,176.570,22.267,153.450
C06181=1088.453,274.799,418.722,176.567,22.264,153.450
C06182=1088.448,274.550,418.752,176.565,22.261,153.450
C06183=1088.442,274.302,418.780,176.561,22.258,153.450
C06184=1088.436,274.054,418.809,176.558,22.255,153.450
C06185=1088.431,273.805,418.838,176.555,22.252,153.449
C06186=1088.425,273.557,418.866,176.552,22.250,153.449
C06187=1088.419,273.309,418.895,176.550,22.247,153.449
C06188=1088.414,273.060,418.924,176.547,22.244,153.449
C06189=1088.409,272.812,418.952,176.544,22.241,153.448
C06190=1088.402,272.564,418.981,176.541,22.238,153.448
C06191=1088.396,272.315,419.009,176.538,22.235,153.448
C06192=1088.391,272.067,419.037,176.535,22.232,153.448
C06193=1088.386,271.819,419.067,176.533,22.230,153.448
C06194=1088.380,271.571,419.095,176.530,22.226,153.447
C06195=1088.374,271.323,419.124,176.527,22.223,153.447
C06196=1088.368,271.074,419.152,176.523,22.221,153.447
C06197=1088.363,270.826,419.180,176.520,22.217,153.447
C06198=1088.357,270.577,419.210,176.517,22.215,153.447
C06199=1088.352,270.329,419.238,176.515,22.212,153.446
C06200=1088.346,270.081,419.266,176.512,22.209,153.446
C06201=1088.341,269.832,419.294,176.509,22.206,153.446
C06202=1088.334,269.584,419.323,176.506,22.203,153.446
C06203=1088.328,269.336,419.352,176.503,22.200,153.446
C06204=1088.323,269.088,419.380,176.501,22.198,153.445
C06205=1088.317,268.839,419.408,176.498,22.195,153.445
C06206=1088.311,268.591,419.437,176.495,22.192,153.445
C06207=1088.305,268.343,419.465,176.492,22.189,153.445
C06208=1088.300,268.095,419.493,176.488,22.186,153.445
C06209=1088.295,267.846,419.522,176.486,22.183,153.444
C06210=1088.290,267.597,419.550,176.483,22.181,153.444
C06211=1088.283,267.349,419.579,176.480,22.178,153.444
C06212=1088.278,267.101,419.607,176.477,22.174,153.444
C06213=1088.272,266.853,419.635,176.474,22.172,153.444
C06214=1088.267,266.604,419.663,176.472,22.169,153.443
C06215=1088.261,266.356,419.691,176.469,22.167,153.443
C06216=1088.255,266.108,419.719,176.466,22.163,153.443
C06217=1088.249,265.859,419.748,176.463,22.160,153.443
C06218=1088.244,265.611,419.776,176.460,22.158,153.443
C06219=1088.238,265.362,419.804,176.457,22.155,153.442
C06220=1088.233,265.114,419.832,176.454,22.152,153.442
C06221=1088.227,264.865,419.860,176.451,22.149,153.442
C06222=1088.222,264.617,419.888,176.448,22.146,153.442
C06223=1088.216,264.369,419.916,176.446,22.144,153.442
C06224=1088.210,264.121,419.944,176.443,22.141,153.441
C06225=1088.204,263.872,419.972,176.440,22.138,153.441
C06226=1088.198,263.624,420.000,176.437,22.135,153.441
C06227=1088.190,263.253,420.042,176.433,22.131,153.441
C06228=1088.180,262.881,420.084,176.428,22.127,153.441
C06229=1088.172,262.510,420.126,176.424,22.123,153.440
C06230=1088.164,262.139,420.167,176.420,22.119,153.440
C06231=1088.157,261.890,420.195,176.417,22.116,153.440
C06232=1088.152,261.642,420.223,176.414,22.113,153.440
C06233=1088.146,261.393,420.251,176.412,22.110,153.439
C06234=1088.140,261.145,420.278,176.408,22.108,153.439
C06235=1088.134,260.896,420.306,176.405,22.105,153.439
C06236=1088.129,260.648,420.334,176.402,22.102,153.439
C06237=1088.124,260.400,420.362,176.400,22.100,153.439
C06238=1088.117,260.151,420.389,176.397,22.097,153.439
C06239=1088.112,259.903,420.417,176.394,22.094,153.439
C06240=1088.106,259.654,420.445,176.391,22.091,153.438
C06241=1088.100,259.407,420.473,176.389,22.088,153.438
C06242=1088.095,259.158,420.500,176.385,22.086,153.438
C06243=1088.089,258.909,420.528,176.382,22.083,153.438
C06244=1088.083,258.661,420.556,176.379,22.080,153.438
C06245=1088.077,258.412,420.583,176.377,22.078,153.437
C06246=1088.072,258.164,420.611,176.374,22.075,153.437
C06247=1088.066,257.916,420.639,176.371,22.072,153.437
C06248=1088.060,257.667,420.666,176.368,22.069,153.437
C06249=1088.054,257.419,420.694,176.366,22.067,153.437
C06250=1088.049,257.170,420.721,176.362,22.064,153.437
C06251=1088.043,256.922,420.749,176.359,22.061,153.436
C06252=1088.037,256.673,420.776,176.357,22.059,153.436
C06253=1088.032,256.425,420.804,176.354,22.056,153.436
C06254=1088.025,256.177,420.831,176.351,22.052,153.436
C06255=1088.020,255.928,420.859,176.348,22.050,153.436
C06256=1088.015,255.680,420.887,176.346,22.047,153.435
C06257=1088.009,255.432,420.913,176.343,22.045,153.435
C06258=1088.003,255.182,420.941,176.339,22.042,153.435
C06259=1087.997,254.935,420.968,176.337,22.039,153.435
C06260=1087.992,254.686,420.996,176.334,22.037,153.435
C06261=1087.987,254.438,421.023,176.331,22.033,153.435
C06262=1087.981,254.189,421.050,176.328,22.030,153.434
C06263=1087.975,253.941,421.078,176.326,22.028,153.434
C06264=1087.969,253.692,421.105,176.323,22.025,153.434
C06265=1087.964,253.444,421.132,176.320,22.022,153.434
C06266=1087.958,253.195,421.160,176.317,22.020,153.434
C06267=1087.953,252.947,421.187,176.314,22.017,153.433
C06268=1087.947,252.698,421.214,176.311,22.014,153.433
C06269=1087.942,252.450,421.242,176.309,22.012,153.433
C06270=1087.936,252.202,421.269,176.306,22.009,153.433
C06271=1087.930,251.953,421.296,176.303,22.006,153.433
C06272=1087.924,251.705,421.324,176.300,22.003,153.433
C06273=1087.919,251.456,421.351,176.298,22.000,153.432
C06274=1087.913,251.208,421.377,176.295,21.998,153.432
C06275=1087.908,250.959,421.405,176.291,21.995,153.432
C06276=1087.902,250.711,421.432,176.289,21.992,153.432
C06277=1087.897,250.462,421.460,176.286,21.990,153.432
C06278=1087.891,250.214,421.486,176.283,21.986,153.432
C06279=1087.883,249.839,421.527,176.279,21.983,153.431
C06280=1087.875,249.466,421.568,176.275,21.978,153.431
C06281=1087.866,249.091,421.609,176.271,21.975,153.431
C06282=1087.857,248.717,421.650,176.266,21.970,153.430
C06283=1087.852,248.468,421.677,176.264,21.968,153.430
C06284=1087.847,248.220,421.703,176.261,21.965,153.430
C06285=1087.842,247.971,421.731,176.258,21.962,153.430
C06286=1087.836,247.723,421.757,176.255,21.959,153.430
C06287=1087.831,247.474,421.785,176.253,21.956,153.430
C06288=1087.825,247.226,421.811,176.250,21.953,153.429
C06289=1087.819,246.977,421.838,176.248,21.951,153.429
C06290=1087.814,246.728,421.865,176.244,21.948,153.429
C06291=1087.808,246.480,421.892,176.241,21.946,153.429
C06292=1087.802,246.232,421.919,176.239,21.943,153.429
C06293=1087.796,245.983,421.945,176.236,21.940,153.429
C06294=1087.791,245.734,421.973,176.233,21.938,153.428
C06295=1087.785,245.486,421.999,176.231,21.935,153.428
C06296=1087.780,245.238,422.026,176.227,21.932,153.428
C06297=1087.774,244.989,422.053,176.225,21.929,153.428
C06298=1087.769,244.741,422.080,176.222,21.927,153.428
C06299=1087.763,244.492,422.107,176.219,21.924,153.428
C06300=1087.757,244.244,422.133,176.216,21.921,153.427
C06301=1087.752,243.996,422.160,176.214,21.919,153.427
C06302=1087.746,243.747,422.186,176.211,21.916,153.427
C06303=1087.741,243.498,422.213,176.208,21.913,153.427
C06304=1087.735,243.250,422.240,176.205,21.911,153.427
C06305=1087.730,243.001,422.266,176.202,21.908,153.427
C06306=1087.723,242.752,422.293,176.200,21.906,153.426
C06307=1087.718,242.503,422.319,176.197,21.903,153.426
C06308=1087.712,242.255,422.346,176.194,21.900,153.426
C06309=1087.706,242.007,422.373,176.192,21.898,153.426
C06310=1087.700,241.758,422.399,176.189,21.895,153.426
C06311=1087.695,241.510,422.426,176.185,21.892,153.426
C06312=1087.689,241.261,422.452,176.183,21.890,153.426
C06313=1087.683,241.012,422.478,176.180,21.887,153.425
C06314=1087.678,240.764,422.505,176.178,21.884,153.425
C06315=1087.672,240.515,422.531,176.175,21.882,153.425
C06316=1087.667,240.266,422.558,176.172,21.879,153.425
C06317=1087.661,240.018,422.585,176.169,21.876,153.425
C06318=1087.656,239.769,422.611,176.166,21.874,153.425
C06319=1087.649,239.521,422.637,176.163,21.871,153.425
C06320=1087.644,239.273,422.664,176.161,21.868,153.424
C06321=1087.638,239.024,422.689,176.158,21.866,153.424
C06322=1087.632,238.775,422.716,176.156,21.863,153.424
C06323=1087.627,238.527,422.742,176.153,21.860,153.424
C06324=1087.622,238.279,422.768,176.149,21.858,153.424
C06325=1087.616,238.030,422.794,176.147,21.855,153.424
C06326=1087.610,237.781,422.821,176.144,21.852,153.423
C06327=1087.605,237.533,422.848,176.142,21.850,153.423
C06328=1087.599,237.284,422.873,176.139,21.847,153.423
C06329=1087.593,237.036,422.900,176.136,21.844,153.423
C06330=1087.588,236.787,422.926,176.133,21.842,153.423
C06331=1087.580,236.406,422.966,176.129,21.837,153.422
C06332=1087.570,236.025,423.006,176.125,21.834,153.422
C06333=1087.562,235.644,423.046,176.121,21.829,153.422
C06334=1087.553,235.263,423.086,176.117,21.826,153.422
C06335=1087.548,235.014,423.112,176.114,21.823,153.422
C06336=1087.542,234.765,423.139,176.111,21.820,153.421
C06337=1087.537,234.517,423.165,176.108,21.818,153.421
C06338=1087.531,234.268,423.191,176.106,21.815,153.421
C06339=1087.525,234.019,423.217,176.103,21.812,153.421
C06340=1087.520,233.771,423.242,176.100,21.810,153.421
C06341=1087.514,233.522,423.268,176.098,21.807,153.421
C06342=1087.509,233.274,423.295,176.095,21.804,153.421
C06343=1087.503,233.025,423.321,176.092,21.802,153.420
C06344=1087.497,232.776,423.346,176.089,21.799,153.420
C06345=1087.492,232.527,423.372,176.087,21.797,153.420
C06346=1087.486,232.279,423.399,176.084,21.794,153.420
C06347=1087.481,232.031,423.424,176.081,21.791,153.420
C06348=1087.475,231.782,423.450,176.079,21.789,153.420
C06349=1087.469,231.533,423.476,176.076,21.786,153.419
C06350=1087.463,231.285,423.502,176.073,21.784,153.419
C06351=1087.459,231.036,423.528,176.070,21.781,153.419
C06352=1087.452,230.788,423.553,176.068,21.778,153.419
C06353=1087.447,230.539,423.579,176.065,21.776,153.419
C06354=1087.441,230.290,423.605,176.063,21.773,153.419
C06355=1087.435,230.041,423.630,176.060,21.770,153.419
C06356=1087.430,229.793,423.657,176.057,21.768,153.418
C06357=1087.424,229.545,423.682,176.054,21.765,153.418
C06358=1087.418,229.296,423.708,176.051,21.762,153.418
C06359=1087.413,229.047,423.734,176.049,21.760,153.418
C06360=1087.407,228.798,423.759,176.046,21.758,153.418
C06361=1087.402,228.550,423.785,176.043,21.755,153.418
C06362=1087.396,228.301,423.810,176.040,21.752,153.418
C06363=1087.390,228.052,423.836,176.038,21.750,153.417
C06364=1087.384,227.803,423.861,176.035,21.747,153.417
C06365=1087.379,227.555,423.887,176.033,21.745,153.417
C06366=1087.373,227.307,423.912,176.030,21.742,153.417
C06367=1087.367,227.058,423.938,176.027,21.740,153.417
C06368=1087.361,226.809,423.964,176.024,21.737,153.417
C06369=1087.356,226.561,423.989,176.021,21.734,153.417
C06370=1087.350,226.312,424.014,176.019,21.732,153.416
C06371=1087.345,226.063,424.040,176.016,21.729,153.416
C06372=1087.340,225.815,424.066,176.014,21.726,153.416
C06373=1087.334,225.566,424.091,176.011,21.724,153.416
C06374=1087.328,225.317,424.117,176.008,21.721,153.416
C06375=1087.323,225.069,424.142,176.005,21.718,153.416
C06376=1087.316,224.820,424.168,176.003,21.716,153.415
C06377=1087.311,224.571,424.193,176.000,21.713,153.415
C06378=1087.306,224.323,424.218,175.998,21.711,153.415
C06379=1087.300,224.074,424.244,175.995,21.708,153.415
C06380=1087.294,223.825,424.269,175.993,21.706,153.415
C06381=1087.289,223.577,424.295,175.989,21.703,153.415
C06382=1087.283,223.328,424.320,175.987,21.701,153.415
C06383=1087.274,222.938,424.359,175.983,21.696,153.414
C06384=1087.266,222.549,424.399,175.979,21.692,153.414
C06385=1087.257,222.159,424.439,175.974,21.688,153.414
C06386=1087.249,221.769,424.478,175.970,21.684,153.414
C06387=1087.243,221.520,424.503,175.967,21.682,153.414
C06388=1087.236,221.272,424.528,175.965,21.679,153.413
C06389=1087.232,221.023,424.554,175.962,21.676,153.413
C06390=1087.226,220.774,424.579,175.960,21.675,153.413
C06391=1087.219,220.525,424.604,175.956,21.672,153.413
C06392=1087.214,220.277,424.629,175.954,21.669,153.413
C06393=1087.209,220.028,424.654,175.951,21.666,153.413
C06394=1087.203,219.780,424.679,175.949,21.664,153.413
C06395=1087.197,219.531,424.704,175.946,21.661,153.412
C06396=1087.191,219.282,424.729,175.944,21.659,153.412
C06397=1087.186,219.034,424.755,175.941,21.656,153.412
C06398=1087.180,218.784,424.779,175.938,21.654,153.412
C06399=1087.175,218.536,424.804,175.935,21.651,153.412
C06400=1087.169,218.287,424.829,175.933,21.648,153.412
C06401=1087.164,218.039,424.854,175.931,21.647,153.412
C06402=1087.158,217.790,424.879,175.928,21.644,153.412
C06403=1087.152,217.542,424.904,175.925,21.641,153.411
C06404=1087.146,217.292,424.929,175.922,21.639,153.411
C06405=1087.140,217.044,424.954,175.920,21.636,153.411
C06406=1087.135,216.795,424.978,175.917,21.633,153.411
C06407=1087.129,216.546,425.004,175.915,21.631,153.411
C06408=1087.124,216.297,425.028,175.912,21.628,153.411
C06409=1087.118,216.049,425.054,175.909,21.626,153.410
C06410=1087.113,215.800,425.078,175.906,21.623,153.410
C06411=1087.107,215.552,425.103,175.904,21.621,153.410
C06412=1087.101,215.303,425.128,175.901,21.618,153.410
C06413=1087.097,215.054,425.152,175.899,21.615,153.410
C06414=1087.090,214.805,425.178,175.897,21.613,153.410
C06415=1087.085,214.557,425.202,175.894,21.610,153.410
C06416=1087.079,214.308,425.227,175.891,21.608,153.409
C06417=1087.074,214.060,425.252,175.888,21.605,153.409
C06418=1087.068,213.810,425.276,175.886,21.602,153.409
C06419=1087.062,213.562,425.300,175.883,21.600,153.409
C06420=1087.057,213.313,425.326,175.881,21.597,153.409
C06421=1087.052,213.064,425.351,175.877,21.595,153.409
C06422=1087.046,212.816,425.375,175.875,21.593,153.409
C06423=1087.040,212.567,425.400,175.873,21.590,153.408
C06424=1087.035,212.318,425.424,175.870,21.587,153.408
C06425=1087.029,212.069,425.449,175.868,21.585,153.408
C06426=1087.024,211.820,425.473,175.865,21.582,153.408
C06427=1087.017,211.572,425.499,175.862,21.580,153.408
C06428=1087.012,211.323,425.523,175.859,21.577,153.408
C06429=1087.007,211.075,425.547,175.857,21.575,153.408
C06430=1087.001,210.825,425.572,175.854,21.572,153.407
C06431=1086.995,210.577,425.595,175.852,21.569,153.407
C06432=1086.989,210.328,425.620,175.849,21.567,153.407
C06433=1086.983,210.080,425.645,175.846,21.565,153.407
C06434=1086.978,209.831,425.669,175.844,21.562,153.407
C06435=1086.969,209.445,425.707,175.839,21.558,153.407
C06436=1086.961,209.059,425.745,175.836,21.554,153.407
C06437=1086.952,208.674,425.783,175.832,21.550,153.406
C06438=1086.944,208.287,425.821,175.828,21.547,153.406
C06439=1086.920,207.262,425.919,175.750,21.506,153.410
C06440=1086.914,207.012,425.944,175.748,21.504,153.410
C06441=1086.909,206.764,425.968,175.745,21.503,153.410
C06442=1086.903,206.515,425.991,175.742,21.501,153.410
C06443=1086.898,206.266,426.015,175.739,21.500,153.410
C06444=1086.893,206.018,426.039,175.737,21.498,153.410
C06445=1086.886,205.769,426.063,175.734,21.497,153.410
C06446=1086.881,205.519,426.087,175.731,21.495,153.410
C06447=1086.875,205.271,426.110,175.729,21.493,153.410
C06448=1086.870,205.023,426.135,175.726,21.491,153.410
C06449=1086.865,204.773,426.158,175.723,21.490,153.410
C06450=1086.859,204.525,426.182,175.720,21.488,153.410
C06451=1086.854,204.276,426.205,175.718,21.487,153.410
C06452=1086.847,204.027,426.229,175.715,21.485,153.411
C06453=1086.842,203.778,426.254,175.713,21.483,153.411
C06454=1086.837,203.529,426.277,175.709,21.482,153.411
C06455=1086.831,203.281,426.301,175.707,21.480,153.411
C06456=1086.826,203.032,426.324,175.704,21.478,153.411
C06457=1086.820,202.783,426.348,175.702,21.477,153.411
C06458=1086.815,202.534,426.372,175.699,21.476,153.411
C06459=1086.809,202.286,426.395,175.697,21.474,153.411
C06460=1086.803,202.036,426.419,175.694,21.472,153.411
C06461=1086.797,201.788,426.443,175.691,21.470,153.411
C06462=1086.791,201.539,426.466,175.688,21.469,153.411
C06463=1086.786,201.290,426.490,175.686,21.467,153.411
C06464=1086.780,201.041,426.513,175.683,21.466,153.411
C06465=1086.775,200.793,426.537,175.680,21.464,153.412
C06466=1086.769,200.544,426.560,175.678,21.463,153.412
C06467=1086.763,200.295,426.584,175.675,21.461,153.412
C06468=1086.758,200.046,426.608,175.673,21.460,153.412
C06469=1086.752,199.797,426.631,175.669,21.458,153.412
C06470=1086.746,199.549,426.654,175.667,21.456,153.412
C06471=1086.741,199.299,426.678,175.664,21.455,153.412
C06472=1086.735,199.051,426.702,175.662,21.453,153.412
C06473=1086.729,198.802,426.725,175.659,21.452,153.412
C06474=1086.724,198.553,426.748,175.656,21.450,153.412
C06475=1086.718,198.305,426.772,175.654,21.449,153.412
C06476=1086.712,198.056,426.795,175.651,21.447,153.412
C06477=1086.707,197.807,426.818,175.649,21.446,153.413
C06478=1086.701,197.557,426.842,175.645,21.443,153.413
C06479=1086.695,197.309,426.865,175.643,21.442,153.413
C06480=1086.689,197.060,426.888,175.640,21.441,153.413
C06481=1086.684,196.811,426.912,175.638,21.439,153.413
C06482=1086.678,196.562,426.935,175.635,21.437,153.413
C06483=1086.672,196.313,426.958,175.633,21.436,153.413
C06484=1086.667,196.064,426.982,175.630,21.434,153.413
C06485=1086.662,195.815,427.005,175.628,21.433,153.413
C06486=1086.656,195.567,427.028,175.625,21.431,153.413
C06487=1086.650,195.318,427.051,175.622,21.429,153.413
C06488=1086.645,195.069,427.075,175.619,21.428,153.413
C06489=1086.639,194.820,427.098,175.616,21.426,153.413
C06490=1086.634,194.571,427.121,175.614,21.424,153.413
C06491=1086.629,194.322,427.144,175.611,21.423,153.414
C06492=1086.623,194.074,427.168,175.609,21.421,153.414
C06493=1086.617,193.825,427.191,175.606,21.420,153.414
C06494=1086.611,193.576,427.214,175.604,21.418,153.414
C06495=1086.606,193.328,427.237,175.601,21.417,153.414
C06496=1086.601,193.078,427.260,175.599,21.415,153.414
C06497=1086.595,192.830,427.283,175.596,21.414,153.414
C06498=1086.589,192.581,427.306,175.594,21.412,153.414
C06499=1086.584,192.332,427.329,175.591,21.410,153.414
C06500=1086.578,192.054,427.355,175.588,21.408,153.414
C06501=1086.571,191.776,427.381,175.585,21.407,153.414
C06502=1086.565,191.498,427.407,175.582,21.405,153.414
C06503=1086.559,191.220,427.432,175.579,21.403,153.414
C06504=1086.553,190.971,427.455,175.577,21.401,153.414
C06505=1086.548,190.722,427.479,175.574,21.399,153.414
C06506=1086.543,190.474,427.501,175.572,21.398,153.415
C06507=1086.537,190.225,427.524,175.569,21.397,153.415
C06508=1086.531,189.976,427.547,175.567,21.395,153.415
C06509=1086.526,189.727,427.570,175.564,21.393,153.415
C06510=1086.521,189.478,427.594,175.562,21.392,153.415
C06511=1086.515,189.229,427.617,175.558,21.390,153.415
C06512=1086.509,188.980,427.640,175.556,21.388,153.415
C06513=1086.504,188.732,427.662,175.553,21.386,153.415
C06514=1086.498,188.483,427.685,175.550,21.385,153.415
C06515=1086.493,188.234,427.707,175.548,21.383,153.415
C06516=1086.488,187.984,427.731,175.545,21.382,153.415
C06517=1086.482,187.735,427.754,175.543,21.380,153.415
C06518=1086.477,187.487,427.777,175.540,21.378,153.415
C06519=1086.471,187.238,427.799,175.538,21.377,153.415
C06520=1086.466,186.989,427.822,175.535,21.375,153.415
C06521=1086.460,186.741,427.845,175.533,21.373,153.415
C06522=1086.455,186.491,427.867,175.530,21.372,153.415
C06523=1086.449,186.243,427.890,175.528,21.370,153.415
C06524=1086.444,185.994,427.914,175.525,21.369,153.416
C06525=1086.439,185.745,427.936,175.523,21.367,153.416
C06526=1086.433,185.495,427.959,175.520,21.365,153.416
C06527=1086.428,185.246,427.982,175.518,21.363,153.416
C06528=1086.422,184.998,428.004,175.515,21.362,153.416
C06529=1086.417,184.749,428.027,175.513,21.360,153.416
C06530=1086.411,184.500,428.049,175.510,21.359,153.416
C06531=1086.405,184.251,428.072,175.508,21.357,153.416
C06532=1086.399,184.002,428.095,175.505,21.356,153.416
C06533=1086.393,183.753,428.118,175.503,21.354,153.416
C06534=1086.387,183.504,428.139,175.500,21.353,153.416
C06535=1086.382,183.256,428.162,175.497,21.351,153.416
C06536=1086.376,183.007,428.185,175.495,21.349,153.416
C06537=1086.371,182.757,428.207,175.492,21.348,153.416
C06538=1086.364,182.509,428.229,175.490,21.347,153.416
C06539=1086.359,182.260,428.252,175.487,21.345,153.416
C06540=1086.353,182.010,428.275,175.485,21.343,153.417
C06541=1086.348,181.762,428.297,175.482,21.342,153.417
C06542=1086.342,181.513,428.319,175.480,21.340,153.417
C06543=1086.336,181.264,428.342,175.477,21.339,153.417
C06544=1086.331,181.015,428.365,175.475,21.337,153.417
C06545=1086.324,180.766,428.386,175.472,21.335,153.417
C06546=1086.319,180.518,428.409,175.470,21.334,153.417
C06547=1086.314,180.268,428.431,175.467,21.333,153.417
C06548=1086.308,180.019,428.454,175.464,21.331,153.417
C06549=1086.302,179.770,428.476,175.462,21.329,153.417
C06550=1086.296,179.521,428.499,175.459,21.327,153.417
C06551=1086.291,179.273,428.521,175.457,21.326,153.417
C06552=1086.285,179.024,428.543,175.454,21.325,153.417
C06553=1086.279,178.774,428.565,175.452,21.323,153.417
C06554=1086.274,178.526,428.588,175.449,21.321,153.418
C06555=1086.268,178.277,428.609,175.447,21.320,153.418
C06556=1086.262,178.028,428.632,175.444,21.318,153.418
C06557=1086.257,177.779,428.654,175.442,21.317,153.418
C06558=1086.251,177.530,428.676,175.439,21.315,153.418
C06559=1086.246,177.281,428.699,175.437,21.313,153.418
C06560=1086.240,177.032,428.721,175.434,21.312,153.418
C06561=1086.234,176.783,428.743,175.432,21.311,153.418
C06562=1086.229,176.534,428.765,175.430,21.309,153.418
C06563=1086.223,176.285,428.787,175.427,21.307,153.418
C06564=1086.216,176.007,428.812,175.424,21.305,153.418
C06565=1086.210,175.729,428.837,175.422,21.304,153.418
C06566=1086.204,175.451,428.862,175.419,21.302,153.418
C06567=1086.198,175.173,428.886,175.416,21.300,153.418
C06568=1086.193,174.923,428.909,175.414,21.298,153.418
C06569=1086.186,174.674,428.930,175.411,21.297,153.418
C06570=1086.181,174.426,428.953,175.409,21.295,153.418
C06571=1086.176,174.177,428.975,175.406,21.294,153.418
C06572=1086.170,173.928,428.996,175.404,21.292,153.418
C06573=1086.165,173.678,429.019,175.401,21.290,153.419
C06574=1086.158,173.430,429.041,175.399,21.289,153.419
C06575=1086.154,173.181,429.063,175.396,21.287,153.419
C06576=1086.147,172.932,429.084,175.394,21.285,153.419
C06577=1086.142,172.682,429.107,175.391,21.284,153.419
C06578=1086.137,172.434,429.129,175.389,21.282,153.419
C06579=1086.131,172.185,429.151,175.386,21.281,153.419
C06580=1086.126,171.936,429.173,175.384,21.279,153.419
C06581=1086.120,171.687,429.194,175.381,21.277,153.419
C06582=1086.115,171.438,429.216,175.379,21.275,153.419
C06583=1086.109,171.189,429.238,175.377,21.274,153.419
C06584=1086.103,170.940,429.261,175.375,21.273,153.419
C06585=1086.098,170.691,429.283,175.372,21.271,153.419
C06586=1086.092,170.442,429.304,175.370,21.269,153.419
C06587=1086.087,170.193,429.326,175.367,21.267,153.419
C06588=1086.081,169.944,429.348,175.365,21.266,153.419
C06589=1086.076,169.695,429.370,175.362,21.264,153.419
C06590=1086.070,169.446,429.391,175.360,21.262,153.419
C06591=1086.065,169.197,429.413,175.357,21.261,153.419
C06592=1086.059,168.948,429.435,175.355,21.259,153.419
C06593=1086.054,168.699,429.457,175.352,21.258,153.419
C06594=1086.048,168.451,429.479,175.351,21.256,153.419
C06595=1086.043,168.202,429.501,175.348,21.254,153.419
C06596=1086.037,167.953,429.522,175.346,21.253,153.419
C06597=1086.032,167.704,429.544,175.343,21.251,153.419
C06598=1086.026,167.454,429.566,175.341,21.249,153.419
C06599=1086.021,167.206,429.588,175.338,21.248,153.420
C06600=1086.015,166.956,429.609,175.336,21.246,153.420
C06601=1086.010,166.708,429.631,175.334,21.244,153.420
C06602=1086.004,166.458,429.653,175.331,21.242,153.420
C06603=1085.999,166.209,429.674,175.329,21.241,153.420
C06604=1085.993,165.960,429.696,175.327,21.239,153.420
C06605=1085.988,165.711,429.717,175.324,21.238,153.420
C06606=1085.983,165.462,429.739,175.322,21.236,153.420
C06607=1085.977,165.213,429.761,175.320,21.234,153.420
C06608=1085.972,164.964,429.782,175.317,21.233,153.420
C06609=1085.966,164.715,429.804,175.315,21.231,153.420
C06610=1085.961,164.466,429.826,175.312,21.229,153.420
C06611=1085.955,164.217,429.848,175.310,21.227,153.420
C06612=1085.950,163.968,429.869,175.308,21.226,153.420
C06613=1085.944,163.719,429.890,175.306,21.224,153.420
C06614=1085.938,163.470,429.912,175.303,21.222,153.420
C06615=1085.934,163.221,429.933,175.301,21.221,153.420
C06616=1085.928,162.973,429.955,175.298,21.219,153.420
C06617=1085.923,162.723,429.977,175.296,21.217,153.420
C06618=1085.917,162.474,429.997,175.293,21.215,153.420
C06619=1085.912,162.225,430.020,175.291,21.214,153.420
C06620=1085.906,161.976,430.041,175.289,21.212,153.420
C06621=1085.901,161.728,430.062,175.287,21.210,153.420
C06622=1085.896,161.477,430.084,175.285,21.208,153.420
C06623=1085.890,161.229,430.105,175.282,21.207,153.420
C06624=1085.884,160.980,430.127,175.280,21.205,153.420
C06625=1085.878,160.731,430.148,175.277,21.203,153.420
C06626=1085.873,160.482,430.168,175.274,21.202,153.420
C06627=1085.867,160.233,430.190,175.273,21.200,153.420
C06628=1085.861,159.954,430.214,175.270,21.198,153.420
C06629=1085.855,159.676,430.237,175.267,21.197,153.420
C06630=1085.848,159.398,430.262,175.265,21.195,153.420
C06631=1085.842,159.119,430.286,175.262,21.193,153.420
C06632=1085.837,158.870,430.306,175.260,21.192,153.420
C06633=1085.831,158.620,430.328,175.257,21.190,153.420
C06634=1085.826,158.372,430.350,175.255,21.188,153.420
C06635=1085.820,158.123,430.370,175.253,21.187,153.420
C06636=1085.814,157.873,430.392,175.251,21.185,153.420
C06637=1085.809,157.625,430.413,175.248,21.183,153.420
C06638=1085.803,157.376,430.434,175.246,21.182,153.420
C06639=1085.797,157.127,430.455,175.243,21.180,153.420
C06640=1085.792,156.877,430.476,175.241,21.178,153.420
C06641=1085.786,156.629,430.497,175.239,21.176,153.420
C06642=1085.780,156.379,430.518,175.237,21.175,153.421
C06643=1085.776,156.130,430.540,175.234,21.173,153.420
C06644=1085.770,155.881,430.561,175.232,21.171,153.420
C06645=1085.764,155.632,430.582,175.229,21.170,153.421
C06646=1085.759,155.383,430.603,175.227,21.168,153.421
C06647=1085.753,155.134,430.624,175.225,21.166,153.421
C06648=1085.748,154.885,430.645,175.223,21.165,153.421
C06649=1085.742,154.636,430.666,175.220,21.163,153.421
C06650=1085.737,154.387,430.687,175.218,21.161,153.421
C06651=1085.731,154.138,430.708,175.216,21.159,153.421
C06652=1085.725,153.889,430.729,175.214,21.158,153.421
C06653=1085.720,153.640,430.750,175.211,21.157,153.421
C06654=1085.713,153.391,430.770,175.209,21.155,153.421
C06655=1085.708,153.142,430.792,175.207,21.153,153.421
C06656=1085.702,152.893,430.812,175.204,21.151,153.421
C06657=1085.696,152.643,430.833,175.202,21.149,153.421
C06658=1085.691,152.395,430.854,175.200,21.148,153.421
C06659=1085.686,152.145,430.875,175.198,21.146,153.421
C06660=1085.680,151.897,430.896,175.195,21.145,153.421
C06661=1085.674,151.647,430.917,175.193,21.143,153.421
C06662=1085.669,151.398,430.938,175.190,21.141,153.421
C06663=1085.663,151.150,430.959,175.189,21.139,153.421
C06664=1085.658,150.900,430.980,175.186,21.138,153.421
C06665=1085.652,150.651,431.001,175.184,21.136,153.421
C06666=1085.647,150.402,431.022,175.181,21.134,153.421
C06667=1085.641,150.153,431.042,175.180,21.133,153.421
C06668=1085.635,149.904,431.062,175.177,21.131,153.421
C06669=1085.630,149.654,431.083,175.175,21.129,153.421
C06670=1085.624,149.406,431.105,175.172,21.128,153.421
C06671=1085.619,149.157,431.125,175.170,21.126,153.421
C06672=1085.614,148.908,431.146,175.169,21.124,153.421
C06673=1085.608,148.658,431.167,175.166,21.122,153.421
C06674=1085.602,148.409,431.188,175.164,21.121,153.421
C06675=1085.596,148.160,431.208,175.161,21.119,153.421
C06676=1085.591,147.911,431.228,175.159,21.117,153.421
C06677=1085.586,147.662,431.249,175.157,21.116,153.421
C06678=1085.579,147.413,431.271,175.155,21.114,153.421
C06679=1085.573,147.164,431.290,175.152,21.113,153.421
C06680=1085.568,146.915,431.311,175.150,21.111,153.421
C06681=1085.563,146.666,431.332,175.148,21.109,153.421
C06682=1085.556,146.416,431.352,175.146,21.107,153.421
C06683=1085.551,146.167,431.372,175.144,21.105,153.421
C06684=1085.546,145.918,431.393,175.141,21.104,153.421
C06685=1085.540,145.670,431.414,175.139,21.103,153.421
C06686=1085.534,145.421,431.434,175.137,21.101,153.421
C06687=1085.529,145.172,431.455,175.135,21.099,153.421
C06688=1085.523,144.922,431.476,175.132,21.097,153.421
C06689=1085.517,144.673,431.496,175.131,21.095,153.421
C06690=1085.512,144.424,431.516,175.128,21.094,153.421
C06691=1085.507,144.175,431.537,175.126,21.092,153.421
C06692=1085.500,143.896,431.560,175.123,21.090,153.421
C06693=1085.494,143.617,431.583,175.121,21.088,153.421
C06694=1085.488,143.338,431.605,175.118,21.086,153.421
C06695=1085.482,143.060,431.629,175.116,21.084,153.421
C06696=1085.475,142.811,431.649,175.114,21.083,153.421
C06697=1085.470,142.562,431.669,175.111,21.081,153.421
C06698=1085.465,142.312,431.690,175.109,21.079,153.421
C06699=1085.459,142.064,431.710,175.107,21.077,153.421
C06700=1085.453,141.814,431.731,175.105,21.075,153.421
C06701=1085.448,141.565,431.750,175.103,21.074,153.421
C06702=1085.442,141.316,431.770,175.100,21.072,153.421
C06703=1085.437,141.067,431.791,175.098,21.071,153.421
C06704=1085.432,140.818,431.811,175.096,21.069,153.421
C06705=1085.426,140.569,431.831,175.094,21.067,153.421
C06706=1085.420,140.319,431.852,175.092,21.065,153.421
C06707=1085.414,140.070,431.872,175.090,21.064,153.421
C06708=1085.409,139.821,431.893,175.087,21.062,153.421
C06709=1085.403,139.572,431.913,175.085,21.060,153.421
C06710=1085.397,139.323,431.933,175.083,21.058,153.421
C06711=1085.392,139.074,431.954,175.081,21.056,153.421
C06712=1085.387,138.825,431.973,175.079,21.054,153.421
C06713=1085.381,138.575,431.994,175.076,21.053,153.421
C06714=1085.375,138.327,432.014,175.075,21.051,153.421
C06715=1085.370,138.078,432.034,175.072,21.050,153.421
C06716=1085.364,137.829,432.054,175.070,21.048,153.421
C06717=1085.358,137.580,432.074,175.068,21.046,153.421
C06718=1085.352,137.329,432.094,175.066,21.045,153.421
C06719=1085.346,137.081,432.114,175.063,21.043,153.421
C06720=1085.341,136.832,432.135,175.061,21.041,153.421
C06721=1085.335,136.583,432.155,175.059,21.039,153.421
C06722=1085.330,136.333,432.175,175.057,21.037,153.421
C06723=1085.324,136.084,432.195,175.055,21.035,153.421
C06724=1085.319,135.835,432.215,175.053,21.034,153.421
C06725=1085.313,135.586,432.235,175.051,21.032,153.421
C06726=1085.307,135.337,432.254,175.048,21.030,153.421
C06727=1085.302,135.088,432.275,175.046,21.028,153.421
C06728=1085.296,134.839,432.295,175.044,21.027,153.421
C06729=1085.291,134.590,432.315,175.042,21.025,153.421
C06730=1085.285,134.340,432.335,175.040,21.023,153.421
C06731=1085.279,134.092,432.355,175.038,21.022,153.420
C06732=1085.274,133.842,432.375,175.036,21.020,153.420
C06733=1085.268,133.593,432.394,175.033,21.018,153.420
C06734=1085.263,133.344,432.415,175.031,21.016,153.420
C06735=1085.257,133.094,432.434,175.029,21.014,153.420
C06736=1085.251,132.846,432.454,175.027,21.013,153.420
C06737=1085.246,132.596,432.475,175.025,21.011,153.420
C06738=1085.240,132.347,432.494,175.023,21.009,153.420
C06739=1085.235,132.098,432.515,175.021,21.007,153.420
C06740=1085.229,131.849,432.534,175.018,21.005,153.420
C06741=1085.223,131.600,432.554,175.017,21.004,153.420
C06742=1085.217,131.351,432.574,175.014,21.002,153.420
C06743=1085.212,131.101,432.593,175.012,21.000,153.420
C06744=1085.206,130.852,432.613,175.010,20.999,153.420
C06745=1085.201,130.603,432.633,175.008,20.997,153.420
C06746=1085.195,130.354,432.653,175.006,20.995,153.420
C06747=1085.189,130.105,432.672,175.004,20.993,153.420
C06748=1085.183,129.856,432.692,175.002,20.992,153.420
C06749=1085.177,129.606,432.711,174.999,20.990,153.420
C06750=1085.172,129.357,432.732,174.997,20.988,153.420
C06751=1085.166,129.108,432.751,174.995,20.986,153.420
C06752=1085.160,128.859,432.771,174.993,20.984,153.420
C06753=1085.155,128.610,432.790,174.991,20.982,153.420
C06754=1085.149,128.361,432.810,174.989,20.981,153.420
C06755=1085.143,128.111,432.829,174.987,20.979,153.420
C06756=1085.137,127.833,432.852,174.984,20.977,153.420
C06757=1085.131,127.554,432.874,174.982,20.975,153.420
C06758=1085.125,127.274,432.896,174.980,20.973,153.420
C06759=1085.118,126.996,432.917,174.977,20.971,153.420
C06760=1085.112,126.747,432.937,174.976,20.970,153.420
C06761=1085.106,126.498,432.957,174.973,20.968,153.420
C06762=1085.101,126.248,432.976,174.971,20.966,153.420
C06763=1085.095,125.999,432.995,174.970,20.964,153.420
C06764=1085.090,125.750,433.016,174.967,20.962,153.420
C06765=1085.085,125.501,433.035,174.965,20.960,153.420
C06766=1085.079,125.252,433.054,174.963,20.959,153.420
C06767=1085.073,125.003,433.074,174.961,20.957,153.420
C06768=1085.067,124.754,433.093,174.958,20.955,153.420
C06769=1085.062,124.504,433.112,174.957,20.954,153.420
C06770=1085.056,124.255,433.132,174.955,20.952,153.420
C06771=1085.050,124.006,433.151,174.952,20.950,153.420
C06772=1085.044,123.756,433.171,174.951,20.948,153.419
C06773=1085.039,123.508,433.190,174.948,20.946,153.419
C06774=1085.033,123.259,433.210,174.946,20.944,153.419
C06775=1085.027,123.009,433.229,174.945,20.943,153.419
C06776=1085.022,122.760,433.248,174.942,20.941,153.419
C06777=1085.017,122.511,433.269,174.940,20.939,153.419
C06778=1085.011,122.261,433.288,174.938,20.937,153.419
C06779=1085.006,122.013,433.307,174.936,20.935,153.419
C06780=1085.000,121.763,433.326,174.934,20.933,153.419
C06781=1084.994,121.514,433.345,174.932,20.932,153.419
C06782=1084.988,121.265,433.365,174.930,20.930,153.419
C06783=1084.983,121.016,433.384,174.928,20.928,153.419
C06784=1084.978,120.767,433.403,174.926,20.926,153.419
C06785=1084.972,120.517,433.422,174.924,20.924,153.419
C06786=1084.966,120.268,433.442,174.922,20.923,153.419
C06787=1084.961,120.019,433.461,174.920,20.921,153.419
C06788=1084.955,119.770,433.481,174.917,20.919,153.419
C06789=1084.949,119.521,433.500,174.916,20.917,153.419
C06790=1084.944,119.272,433.519,174.914,20.915,153.419
C06791=1084.938,119.022,433.538,174.911,20.913,153.419
C06792=1084.932,118.773,433.558,174.910,20.912,153.419
C06793=1084.927,118.524,433.576,174.908,20.909,153.418
C06794=1084.922,118.275,433.596,174.906,20.908,153.418
C06795=1084.916,118.025,433.615,174.904,20.906,153.418
C06796=1084.910,117.776,433.634,174.901,20.904,153.418
C06797=1084.905,117.527,433.653,174.900,20.902,153.418
C06798=1084.899,117.278,433.672,174.898,20.900,153.418
C06799=1084.894,117.028,433.692,174.895,20.898,153.418
C06800=1084.889,116.779,433.710,174.894,20.896,153.418
C06801=1084.883,116.530,433.730,174.892,20.894,153.418
C06802=1084.877,116.280,433.749,174.890,20.893,153.418
C06803=1084.872,116.032,433.768,174.888,20.891,153.418
C06804=1084.867,115.782,433.787,174.885,20.888,153.418
C06805=1084.861,115.533,433.806,174.884,20.887,153.418
C06806=1084.856,115.284,433.825,174.882,20.885,153.418
C06807=1084.850,115.035,433.844,174.880,20.883,153.417
C06808=1084.844,114.785,433.864,174.878,20.881,153.417
C06809=1084.839,114.537,433.882,174.875,20.879,153.417
C06810=1084.833,114.287,433.901,174.874,20.877,153.417
C06811=1084.827,114.038,433.920,174.872,20.875,153.417
C06812=1084.822,113.789,433.940,174.869,20.874,153.417
C06813=1084.816,113.540,433.958,174.868,20.872,153.417
C06814=1084.810,113.291,433.977,174.866,20.870,153.417
C06815=1084.804,113.041,433.996,174.864,20.868,153.417
C06816=1084.799,112.793,434.015,174.862,20.866,153.417
C06817=1084.794,112.543,434.034,174.860,20.864,153.417
C06818=1084.788,112.293,434.053,174.858,20.862,153.417
C06819=1084.782,112.045,434.071,174.856,20.860,153.417
C06820=1084.776,111.765,434.093,174.854,20.858,153.417
C06821=1084.769,111.486,434.114,174.851,20.856,153.417
C06822=1084.763,111.207,434.135,174.850,20.854,153.417
C06823=1084.757,110.928,434.156,174.847,20.852,153.417
C06824=1084.752,110.680,434.175,174.845,20.850,153.416
C06825=1084.745,110.430,434.194,174.843,20.848,153.416
C06826=1084.740,110.180,434.212,174.841,20.846,153.416
C06827=1084.735,109.932,434.231,174.839,20.845,153.416
C06828=1084.728,109.683,434.250,174.837,20.843,153.416
C06829=1084.723,109.433,434.269,174.835,20.841,153.416
C06830=1084.717,109.185,434.287,174.834,20.839,153.416
C06831=1084.711,108.935,434.306,174.831,20.837,153.416
C06832=1084.706,108.685,434.325,174.829,20.835,153.416
C06833=1084.700,108.437,434.343,174.828,20.833,153.416
C06834=1084.695,108.187,434.362,174.825,20.832,153.416
C06835=1084.688,107.938,434.380,174.824,20.830,153.416
C06836=1084.683,107.689,434.399,174.822,20.828,153.416
C06837=1084.677,107.439,434.419,174.820,20.826,153.416
C06838=1084.671,107.190,434.436,174.818,20.824,153.415
C06839=1084.666,106.941,434.455,174.816,20.822,153.415
C06840=1084.660,106.692,434.474,174.814,20.820,153.415
C06841=1084.655,106.442,434.492,174.812,20.818,153.415
C06842=1084.649,106.193,434.511,174.810,20.817,153.415
C06843=1084.643,105.943,434.529,174.808,20.815,153.415
C06844=1084.638,105.695,434.548,174.806,20.812,153.415
C06845=1084.632,105.445,434.567,174.804,20.811,153.415
C06846=1084.627,105.196,434.585,174.802,20.808,153.415
C06847=1084.620,104.947,434.604,174.801,20.807,153.415
C06848=1084.616,104.698,434.622,174.798,20.805,153.415
C06849=1084.610,104.448,434.641,174.797,20.803,153.415
C06850=1084.604,104.199,434.660,174.795,20.801,153.415
C06851=1084.599,103.950,434.678,174.793,20.799,153.414
C06852=1084.592,103.701,434.697,174.791,20.797,153.414
C06853=1084.588,103.451,434.715,174.789,20.795,153.414
C06854=1084.581,103.202,434.733,174.787,20.793,153.414
C06855=1084.576,102.953,434.751,174.785,20.791,153.414
C06856=1084.570,102.704,434.770,174.783,20.789,153.414
C06857=1084.565,102.454,434.788,174.781,20.788,153.414
C06858=1084.559,102.205,434.807,174.780,20.786,153.414
C06859=1084.554,101.956,434.825,174.777,20.784,153.414
C06860=1084.548,101.706,434.844,174.775,20.781,153.414
C06861=1084.543,101.457,434.862,174.774,20.780,153.414
C06862=1084.537,101.208,434.881,174.772,20.777,153.414
C06863=1084.532,100.959,434.899,174.770,20.776,153.414
C06864=1084.525,100.710,434.917,174.768,20.773,153.413
C06865=1084.520,100.460,434.936,174.766,20.772,153.413
C06866=1084.514,100.211,434.953,174.764,20.770,153.413
C06867=1084.508,99.962,434.972,174.763,20.768,153.413
C06868=1084.503,99.712,434.990,174.760,20.766,153.413
C06869=1084.497,99.463,435.009,174.759,20.764,153.413
C06870=1084.491,99.214,435.027,174.757,20.762,153.413
C06871=1084.486,98.964,435.045,174.754,20.760,153.413
C06872=1084.480,98.716,435.063,174.753,20.758,153.413
C06873=1084.474,98.466,435.081,174.751,20.757,153.413
C06874=1084.469,98.217,435.100,174.749,20.755,153.413
C06875=1084.463,97.967,435.118,174.747,20.753,153.413
C06876=1084.457,97.718,435.136,174.746,20.751,153.412
C06877=1084.451,97.469,435.155,174.743,20.749,153.412
C06878=1084.446,97.220,435.172,174.742,20.747,153.412
C06879=1084.440,96.970,435.190,174.739,20.745,153.412
C06880=1084.434,96.722,435.209,174.738,20.743,153.412
C06881=1084.428,96.472,435.227,174.736,20.741,153.412
C06882=1084.423,96.223,435.245,174.734,20.739,153.412
C06883=1084.417,95.974,435.262,174.732,20.737,153.412
C06884=1084.411,95.695,435.283,174.730,20.735,153.412
C06885=1084.404,95.415,435.303,174.728,20.733,153.412
C06886=1084.398,95.136,435.324,174.726,20.731,153.412
C06887=1084.392,94.858,435.344,174.724,20.728,153.411
C06888=1084.386,94.608,435.362,174.722,20.726,153.411
C06889=1084.381,94.359,435.380,174.720,20.725,153.411
C06890=1084.375,94.110,435.398,174.718,20.723,153.411
C06891=1084.369,93.861,435.416,174.717,20.721,153.411
C06892=1084.364,93.612,435.434,174.715,20.718,153.411
C06893=1084.358,93.362,435.452,174.713,20.717,153.411
C06894=1084.353,93.113,435.470,174.711,20.714,153.411
C06895=1084.346,92.863,435.488,174.709,20.713,153.411
C06896=1084.341,92.614,435.506,174.707,20.710,153.411
C06897=1084.336,92.365,435.524,174.705,20.708,153.411
C06898=1084.330,92.115,435.542,174.704,20.707,153.410
C06899=1084.325,91.866,435.560,174.701,20.704,153.410
C06900=1084.319,91.617,435.577,174.700,20.703,153.410
C06901=1084.313,91.368,435.595,174.698,20.700,153.410
C06902=1084.308,91.119,435.614,174.696,20.699,153.410
C06903=1084.302,90.869,435.632,174.694,20.696,153.410
C06904=1084.296,90.620,435.649,174.693,20.695,153.410
C06905=1084.291,90.371,435.667,174.690,20.692,153.410
C06906=1084.285,90.121,435.685,174.689,20.691,153.410
C06907=1084.279,89.872,435.703,174.687,20.689,153.409
C06908=1084.273,89.622,435.720,174.685,20.687,153.409
C06909=1084.267,89.373,435.738,174.683,20.685,153.409
C06910=1084.262,89.124,435.756,174.682,20.683,153.409
C06911=1084.256,88.875,435.774,174.679,20.681,153.409
C06912=1084.250,88.626,435.791,174.678,20.679,153.409
C06913=1084.244,88.376,435.809,174.676,20.677,153.409
C06914=1084.239,88.127,435.827,174.674,20.675,153.409
C06915=1084.233,87.878,435.844,174.672,20.673,153.409
C06916=1084.227,87.628,435.862,174.671,20.671,153.409
C06917=1084.221,87.379,435.880,174.669,20.669,153.408
C06918=1084.216,87.130,435.897,174.667,20.667,153.408
C06919=1084.210,86.880,435.915,174.665,20.665,153.408
C06920=1084.204,86.631,435.933,174.663,20.663,153.408
C06921=1084.199,86.382,435.950,174.661,20.661,153.408
C06922=1084.193,86.132,435.968,174.660,20.659,153.408
C06923=1084.187,85.883,435.986,174.658,20.657,153.408
C06924=1084.182,85.634,436.003,174.656,20.655,153.408
C06925=1084.175,85.385,436.021,174.654,20.653,153.408
C06926=1084.170,85.135,436.038,174.653,20.651,153.407
C06927=1084.165,84.886,436.056,174.650,20.649,153.407
C06928=1084.159,84.636,436.074,174.649,20.647,153.407
C06929=1084.153,84.387,436.091,174.647,20.645,153.407
C06930=1084.148,84.138,436.109,174.645,20.643,153.407
C06931=1084.142,83.889,436.126,174.643,20.641,153.407
C06932=1084.136,83.639,436.144,174.642,20.639,153.407
C06933=1084.131,83.390,436.161,174.639,20.637,153.407
C06934=1084.125,83.141,436.179,174.638,20.635,153.407
C06935=1084.119,82.891,436.197,174.637,20.633,153.406
C06936=1084.114,82.642,436.214,174.634,20.631,153.406
C06937=1084.108,82.393,436.232,174.633,20.629,153.406
C06938=1084.103,82.144,436.249,174.631,20.627,153.406
C06939=1084.097,81.893,436.267,174.630,20.625,153.406
C06940=1084.091,81.644,436.284,174.627,20.623,153.406
C06941=1084.086,81.395,436.302,174.626,20.621,153.406
C06942=1084.080,81.146,436.319,174.624,20.618,153.406
C06943=1084.075,80.897,436.336,174.622,20.617,153.406
C06944=1084.068,80.647,436.353,174.620,20.614,153.405
C06945=1084.063,80.398,436.371,174.619,20.612,153.405
C06946=1084.057,80.149,436.389,174.617,20.611,153.405
C06947=1084.052,79.899,436.405,174.615,20.609,153.405
C06948=1084.045,79.620,436.425,174.613,20.606,153.405
C06949=1084.039,79.342,436.445,174.611,20.604,153.405
C06950=1084.033,79.063,436.464,174.609,20.601,153.405
C06951=1084.026,78.784,436.484,174.607,20.599,153.404
C06952=1084.021,78.534,436.501,174.605,20.597,153.404
C06953=1084.015,78.285,436.518,174.604,20.595,153.404
C06954=1084.009,78.036,436.535,174.602,20.593,153.404
C06955=1084.004,77.786,436.552,174.600,20.591,153.404
C06956=1083.998,77.537,436.570,174.598,20.589,153.404
C06957=1083.992,77.288,436.588,174.597,20.587,153.404
C06958=1083.987,77.039,436.604,174.595,20.585,153.404
C06959=1083.981,76.790,436.621,174.593,20.583,153.403
C06960=1083.975,76.539,436.639,174.592,20.581,153.403
C06961=1083.969,76.291,436.656,174.590,20.579,153.403
C06962=1083.963,76.041,436.673,174.588,20.577,153.403
C06963=1083.958,75.792,436.690,174.586,20.575,153.403
C06964=1083.953,75.543,436.708,174.585,20.573,153.403
C06965=1083.946,75.293,436.724,174.582,20.570,153.403
C06966=1083.941,75.044,436.742,174.581,20.569,153.403
C06967=1083.935,74.794,436.759,174.579,20.566,153.403
C06968=1083.929,74.545,436.776,174.578,20.565,153.402
C06969=1083.924,74.296,436.792,174.575,20.562,153.402
C06970=1083.918,74.047,436.810,174.574,20.561,153.402
C06971=1083.912,73.797,436.827,174.573,20.559,153.402
C06972=1083.906,73.548,436.844,174.570,20.556,153.402
C06973=1083.901,73.298,436.862,174.569,20.554,153.402
C06974=1083.895,73.049,436.878,174.567,20.552,153.402
C06975=1083.890,72.799,436.895,174.565,20.550,153.402
C06976=1083.884,72.550,436.912,174.563,20.548,153.401
C06977=1083.878,72.301,436.929,174.562,20.546,153.401
C06978=1083.873,72.052,436.946,174.560,20.543,153.401
C06979=1083.867,71.802,436.963,174.558,20.542,153.401
C06980=1083.861,71.553,436.980,174.557,20.540,153.401
C06981=1083.855,71.303,436.997,174.555,20.538,153.401
C06982=1083.850,71.054,437.015,174.554,20.536,153.401
C06983=1083.844,70.805,437.031,174.551,20.534,153.401
C06984=1083.839,70.555,437.048,174.550,20.532,153.400
C06985=1083.832,70.307,437.065,174.548,20.529,153.400
C06986=1083.827,70.057,437.082,174.547,20.527,153.400
C06987=1083.822,69.808,437.099,174.544,20.525,153.400
C06988=1083.815,69.558,437.116,174.543,20.523,153.400
C06989=1083.810,69.308,437.133,174.542,20.521,153.400
C06990=1083.804,69.059,437.150,174.539,20.519,153.400
C06991=1083.798,68.810,437.167,174.538,20.517,153.399
C06992=1083.793,68.560,437.183,174.536,20.514,153.399
C06993=1083.787,68.311,437.200,174.534,20.513,153.399
C06994=1083.781,68.062,437.217,174.532,20.511,153.399
C06995=1083.776,67.812,437.234,174.531,20.509,153.399
C06996=1083.770,67.564,437.251,174.530,20.507,153.399
C06997=1083.764,67.314,437.267,174.528,20.504,153.399
C06998=1083.758,67.065,437.284,174.526,20.503,153.399
C06999=1083.753,66.815,437.301,174.524,20.500,153.398
C07000=1083.747,66.566,437.317,174.523,20.498,153.398
C07001=1083.741,66.316,437.335,174.521,20.496,153.398
C07002=1083.735,66.066,437.351,174.519,20.494,153.398
C07003=1083.729,65.817,437.367,174.518,20.492,153.398
C07004=1083.724,65.568,437.385,174.516,20.490,153.398
C07005=1083.718,65.319,437.401,174.514,20.488,153.398
C07006=1083.713,65.069,437.418,174.512,20.486,153.397
C07007=1083.707,64.820,437.434,174.511,20.484,153.397
C07008=1083.701,64.570,437.451,174.509,20.481,153.397
C07009=1083.695,64.321,437.468,174.507,20.480,153.397
C07010=1083.689,64.072,437.484,174.506,20.478,153.397
C07011=1083.684,63.822,437.501,174.504,20.475,153.397
C07012=1083.677,63.544,437.519,174.502,20.473,153.397
C07013=1083.670,63.265,437.538,174.500,20.471,153.396
C07014=1083.664,62.986,437.557,174.498,20.468,153.396
C07015=1083.658,62.707,437.575,174.496,20.466,153.396
C07016=1083.652,62.457,437.591,174.495,20.464,153.396
C07017=1083.646,62.208,437.608,174.493,20.462,153.396
C07018=1083.640,61.959,437.624,174.491,20.460,153.396
C07019=1083.634,61.710,437.641,174.490,20.458,153.396
C07020=1083.628,61.460,437.658,174.488,20.456,153.395
C07021=1083.623,61.211,437.674,174.486,20.454,153.395
C07022=1083.617,60.961,437.690,174.485,20.452,153.395
C07023=1083.611,60.712,437.707,174.483,20.450,153.395
C07024=1083.605,60.462,437.723,174.481,20.448,153.395
C07025=1083.599,60.213,437.740,174.479,20.445,153.395
C07026=1083.593,59.964,437.756,174.478,20.444,153.395
C07027=1083.588,59.714,437.772,174.476,20.441,153.395
C07028=1083.582,59.465,437.789,174.474,20.439,153.394
C07029=1083.576,59.215,437.805,174.473,20.437,153.394
C07030=1083.570,58.966,437.822,174.471,20.435,153.394
C07031=1083.564,58.717,437.838,174.469,20.433,153.394
C07032=1083.559,58.467,437.854,174.467,20.431,153.394
C07033=1083.553,58.218,437.871,174.466,20.429,153.394
C07034=1083.547,57.968,437.887,174.465,20.427,153.394
C07035=1083.541,57.719,437.903,174.463,20.425,153.393
C07036=1083.535,57.470,437.920,174.461,20.423,153.393
C07037=1083.530,57.220,437.936,174.459,20.420,153.393
C07038=1083.524,56.971,437.952,174.458,20.419,153.393
C07039=1083.518,56.721,437.969,174.456,20.417,153.393
C07040=1083.512,56.472,437.985,174.454,20.414,153.393
C07041=1083.506,56.223,438.002,174.453,20.412,153.393
C07042=1083.500,55.973,438.018,174.452,20.410,153.392
C07043=1083.495,55.724,438.034,174.450,20.408,153.392
C07044=1083.489,55.475,438.050,174.448,20.406,153.392
C07045=1083.484,55.224,438.066,174.446,20.403,153.392
C07046=1083.478,54.976,438.082,174.445,20.402,153.392
C07047=1083.472,54.726,438.099,174.443,20.400,153.392
C07048=1083.466,54.477,438.115,174.441,20.397,153.392
C07049=1083.460,54.228,438.131,174.440,20.395,153.391
C07050=1083.455,53.978,438.147,174.438,20.393,153.391
C07051=1083.449,53.729,438.164,174.436,20.391,153.391
C07052=1083.444,53.479,438.180,174.435,20.389,153.391
C07053=1083.438,53.229,438.196,174.433,20.387,153.391
C07054=1083.432,52.980,438.212,174.432,20.385,153.391
C07055=1083.426,52.731,438.228,174.430,20.382,153.390
C07056=1083.420,52.482,438.244,174.428,20.380,153.390
C07057=1083.415,52.232,438.260,174.427,20.378,153.390
C07058=1083.409,51.983,438.276,174.425,20.376,153.390
C07059=1083.403,51.733,438.292,174.423,20.374,153.390
C07060=1083.398,51.484,438.309,174.422,20.372,153.390
C07061=1083.392,51.234,438.326,174.420,20.370,153.390
C07062=1083.387,50.985,438.341,174.419,20.368,153.389
C07063=1083.381,50.736,438.357,174.417,20.365,153.389
C07064=1083.375,50.486,438.373,174.415,20.363,153.389
C07065=1083.369,50.237,438.390,174.414,20.361,153.389
C07066=1083.363,49.987,438.405,174.412,20.359,153.389
C07067=1083.357,49.738,438.421,174.411,20.357,153.389
C07068=1083.352,49.489,438.437,174.409,20.355,153.388
C07069=1083.346,49.239,438.453,174.407,20.352,153.388
C07070=1083.340,48.990,438.469,174.406,20.351,153.388
C07071=1083.334,48.740,438.485,174.404,20.348,153.388
C07072=1083.329,48.490,438.501,174.402,20.346,153.388
C07073=1083.324,48.241,438.517,174.401,20.344,153.388
C07074=1083.318,47.992,438.534,174.399,20.342,153.387
C07075=1083.313,47.742,438.549,174.398,20.340,153.387
C07076=1083.306,47.463,438.567,174.396,20.337,153.387
C07077=1083.300,47.184,438.585,174.394,20.335,153.387
C07078=1083.293,46.905,438.603,174.392,20.332,153.387
C07079=1083.287,46.626,438.621,174.390,20.330,153.387
C07080=1083.281,46.376,438.636,174.389,20.328,153.386
C07081=1083.276,46.128,438.652,174.388,20.326,153.386
C07082=1083.270,45.878,438.668,174.386,20.323,153.386
C07083=1083.264,45.628,438.684,174.384,20.321,153.386
C07084=1083.259,45.378,438.700,174.382,20.319,153.386
C07085=1083.253,45.130,438.716,174.381,20.317,153.386
C07086=1083.247,44.880,438.732,174.380,20.315,153.385
C07087=1083.242,44.630,438.747,174.377,20.312,153.385
C07088=1083.236,44.382,438.763,174.376,20.310,153.385
C07089=1083.231,44.132,438.779,174.375,20.308,153.385
C07090=1083.225,43.882,438.795,174.373,20.306,153.385
C07091=1083.219,43.632,438.811,174.372,20.304,153.385
C07092=1083.214,43.384,438.826,174.370,20.302,153.384
C07093=1083.208,43.134,438.842,174.368,20.300,153.384
C07094=1083.202,42.884,438.858,174.367,20.298,153.384
C07095=1083.196,42.635,438.873,174.365,20.295,153.384
C07096=1083.190,42.386,438.889,174.363,20.293,153.384
C07097=1083.185,42.136,438.905,174.362,20.291,153.384
C07098=1083.179,41.887,438.921,174.360,20.289,153.384
C07099=1083.173,41.637,438.936,174.359,20.287,153.383
C07100=1083.168,41.388,438.952,174.357,20.285,153.383
C07101=1083.161,41.138,438.967,174.355,20.282,153.383
C07102=1083.156,40.888,438.983,174.354,20.280,153.383
C07103=1083.150,40.640,438.999,174.353,20.278,153.383
C07104=1083.145,40.390,439.014,174.351,20.276,153.383
C07105=1083.139,40.141,439.030,174.349,20.274,153.382
C07106=1083.133,39.892,439.045,174.348,20.272,153.382
C07107=1083.127,39.642,439.061,174.346,20.269,153.382
C07108=1083.121,39.392,439.077,174.345,20.267,153.382
C07109=1083.116,39.143,439.092,174.343,20.265,153.382
C07110=1083.111,38.893,439.108,174.341,20.263,153.382
C07111=1083.104,38.644,439.123,174.340,20.261,153.381
C07112=1083.098,38.394,439.139,174.339,20.259,153.381
C07113=1083.093,38.145,439.154,174.337,20.256,153.381
C07114=1083.087,37.895,439.170,174.335,20.254,153.381
C07115=1083.081,37.646,439.185,174.333,20.252,153.381
C07116=1083.076,37.396,439.200,174.332,20.250,153.381
C07117=1083.070,37.147,439.217,174.331,20.248,153.380
C07118=1083.064,36.897,439.232,174.329,20.246,153.380
C07119=1083.059,36.648,439.247,174.327,20.244,153.380
C07120=1083.053,36.399,439.263,174.326,20.242,153.380
C07121=1083.046,36.149,439.278,174.324,20.239,153.380
C07122=1083.041,35.900,439.293,174.323,20.237,153.380
C07123=1083.035,35.650,439.308,174.321,20.235,153.379
C07124=1083.029,35.401,439.324,174.319,20.233,153.379
C07125=1083.024,35.152,439.339,174.318,20.231,153.379
C07126=1083.017,34.902,439.354,174.317,20.229,153.379
C07127=1083.012,34.652,439.370,174.314,20.226,153.379
C07128=1083.006,34.403,439.386,174.313,20.224,153.379
C07129=1083.000,34.154,439.401,174.312,20.222,153.378
C07130=1082.994,33.904,439.416,174.310,20.220,153.378
C07131=1082.989,33.655,439.431,174.309,20.218,153.378
C07132=1082.983,33.405,439.446,174.307,20.216,153.378
C07133=1082.976,33.156,439.462,174.305,20.213,153.378
C07134=1082.971,32.907,439.477,174.304,20.211,153.378
C07135=1082.966,32.657,439.493,174.303,20.209,153.377
C07136=1082.960,32.408,439.507,174.301,20.207,153.377
C07137=1082.954,32.158,439.523,174.299,20.205,153.377
C07138=1082.948,31.908,439.538,174.298,20.203,153.377
C07139=1082.942,31.659,439.554,174.297,20.201,153.377
C07140=1082.935,31.380,439.571,174.295,20.198,153.377
C07141=1082.929,31.101,439.588,174.293,20.195,153.376
C07142=1082.923,30.822,439.604,174.291,20.193,153.376
C07143=1082.917,30.543,439.622,174.289,20.191,153.376
C07144=1082.910,30.293,439.637,174.288,20.189,153.376
C07145=1082.905,30.044,439.652,174.287,20.187,153.376
C07146=1082.900,29.794,439.667,174.285,20.184,153.376
C07147=1082.894,29.545,439.682,174.283,20.182,153.375
C07148=1082.888,29.295,439.698,174.282,20.180,153.375
C07149=1082.882,29.045,439.713,174.280,20.178,153.375
C07150=1082.877,28.796,439.728,174.279,20.176,153.375
C07151=1082.870,28.546,439.743,174.277,20.174,153.375
C07152=1082.865,28.297,439.758,174.275,20.172,153.375
C07153=1082.859,28.048,439.773,174.274,20.170,153.374
C07154=1082.853,27.799,439.787,174.273,20.168,153.374
C07155=1082.848,27.549,439.803,174.271,20.165,153.374
C07156=1082.841,27.299,439.818,174.269,20.163,153.374
C07157=1082.836,27.050,439.833,174.268,20.161,153.374
C07158=1082.830,26.800,439.848,174.266,20.159,153.374
C07159=1082.824,26.551,439.863,174.265,20.157,153.373
C07160=1082.818,26.301,439.878,174.263,20.155,153.373
C07161=1082.813,26.052,439.893,174.262,20.153,153.373
C07162=1082.807,25.802,439.908,174.260,20.150,153.373
C07163=1082.801,25.553,439.923,174.259,20.148,153.373
C07164=1082.795,25.304,439.938,174.257,20.146,153.373
C07165=1082.790,25.054,439.953,174.255,20.144,153.372
C07166=1082.783,24.805,439.968,174.254,20.142,153.372
C07167=1082.777,24.555,439.983,174.253,20.140,153.372
C07168=1082.772,24.306,439.998,174.251,20.137,153.372
C07169=1082.766,24.055,440.012,174.249,20.135,153.372
C07170=1082.760,23.807,440.027,174.248,20.133,153.372
C07171=1082.754,23.557,440.042,174.246,20.130,153.371
C07172=1082.749,23.308,440.057,174.245,20.128,153.371
C07173=1082.742,23.058,440.072,174.244,20.126,153.371
C07174=1082.737,22.809,440.087,174.242,20.124,153.371
C07175=1082.731,22.559,440.102,174.240,20.122,153.371
C07176=1082.725,22.310,440.117,174.239,20.120,153.371
C07177=1082.720,22.059,440.131,174.238,20.118,153.370
C07178=1082.714,21.810,440.146,174.236,20.115,153.370
C07179=1082.708,21.562,440.161,174.234,20.113,153.370
C07180=1082.702,21.312,440.176,174.233,20.111,153.370
C07181=1082.697,21.063,440.191,174.231,20.109,153.370
C07182=1082.691,20.812,440.205,174.230,20.107,153.370
C07183=1082.686,20.563,440.220,174.228,20.105,153.369
C07184=1082.679,20.313,440.235,174.227,20.103,153.369
C07185=1082.673,20.064,440.250,174.225,20.100,153.369
C07186=1082.667,19.815,440.265,174.224,20.098,153.369
C07187=1082.662,19.565,440.279,174.223,20.096,153.369
C07188=1082.656,19.315,440.294,174.220,20.094,153.369
C07189=1082.650,19.066,440.308,174.219,20.092,153.368
C07190=1082.644,18.816,440.323,174.218,20.090,153.368
C07191=1082.638,18.567,440.337,174.217,20.088,153.368
C07192=1082.633,18.318,440.352,174.214,20.085,153.368
C07193=1082.627,18.068,440.367,174.213,20.083,153.368
C07194=1082.621,17.819,440.381,174.212,20.081,153.368
C07195=1082.615,17.569,440.396,174.210,20.079,153.367
C07196=1082.609,17.320,440.411,174.209,20.077,153.367
C07197=1082.603,17.070,440.425,174.207,20.075,153.367
C07198=1082.598,16.820,440.440,174.206,20.073,153.367
C07199=1082.592,16.571,440.455,174.204,20.070,153.367
C07200=1082.586,16.321,440.469,174.203,20.068,153.367
C07201=1082.580,16.072,440.484,174.201,20.066,153.366
C07202=1082.574,15.823,440.499,174.199,20.064,153.366
C07203=1082.569,15.573,440.512,174.198,20.062,153.366
C07204=1082.562,15.295,440.530,174.197,20.059,153.366
C07205=1082.556,15.017,440.546,174.195,20.057,153.366
C07206=1082.550,14.740,440.561,174.194,20.055,153.365
C07207=1082.543,14.462,440.578,174.191,20.052,153.365
C07208=1082.538,14.213,440.592,174.190,20.050,153.365
C07209=1082.531,13.963,440.607,174.188,20.048,153.365
C07210=1082.526,13.713,440.621,174.187,20.046,153.365
C07211=1082.519,13.464,440.636,174.186,20.044,153.365
C07212=1082.514,13.214,440.650,174.184,20.042,153.365
C07213=1082.508,12.965,440.664,174.182,20.039,153.364
C07214=1082.502,12.716,440.679,174.181,20.037,153.364
C07215=1082.496,12.466,440.693,174.180,20.035,153.364
C07216=1082.490,12.216,440.708,174.178,20.033,153.364
C07217=1082.484,11.967,440.721,174.176,20.031,153.364
C07218=1082.478,11.718,440.736,174.175,20.029,153.364
C07219=1082.472,11.468,440.750,174.174,20.027,153.363
C07220=1082.466,11.219,440.765,174.172,20.025,153.363
C07221=1082.460,10.969,440.779,174.170,20.023,153.363
C07222=1082.454,10.720,440.794,174.169,20.021,153.363
C07223=1082.449,10.470,440.807,174.168,20.019,153.363
C07224=1082.442,10.220,440.822,174.166,20.016,153.363
C07225=1082.437,9.971,440.836,174.164,20.014,153.362
C07226=1082.431,9.721,440.850,174.163,20.012,153.362
C07227=1082.425,9.472,440.865,174.162,20.010,153.362
C07228=1082.419,9.222,440.879,174.160,20.008,153.362
C07229=1082.413,8.972,440.894,174.159,20.006,153.362
C07230=1082.408,8.723,440.908,174.157,20.004,153.362
C07231=1082.402,8.474,440.922,174.156,20.002,153.361
C07232=1082.396,8.224,440.937,174.154,19.999,153.361
C07233=1082.390,7.974,440.950,174.153,19.997,153.361
C07234=1082.384,7.725,440.964,174.151,19.995,153.361
C07235=1082.378,7.476,440.978,174.150,19.993,153.361
C07236=1082.372,7.226,440.993,174.148,19.991,153.361
C07237=1082.366,6.977,441.007,174.147,19.989,153.360
C07238=1082.361,6.727,441.021,174.145,19.987,153.360
C07239=1082.355,6.477,441.036,174.144,19.985,153.360
C07240=1082.349,6.228,441.050,174.142,19.983,153.360
C07241=1082.344,5.978,441.064,174.141,19.981,153.360
C07242=1082.337,5.729,441.079,174.139,19.979,153.360
C07243=1082.331,5.479,441.092,174.137,19.976,153.360
C07244=1082.326,5.230,441.106,174.136,19.974,153.359
C07245=1082.320,4.981,441.120,174.135,19.972,153.359
C07246=1082.314,4.730,441.134,174.133,19.970,153.359
C07247=1082.308,4.481,441.148,174.131,19.968,153.359
C07248=1082.302,4.232,441.163,174.130,19.966,153.359
C07249=1082.297,3.982,441.177,174.129,19.964,153.359
C07250=1082.291,3.732,441.191,174.128,19.962,153.358
C07251=1082.285,3.483,441.204,174.126,19.959,153.358
C07252=1082.279,3.234,441.219,174.124,19.957,153.358
C07253=1082.273,2.984,441.233,174.123,19.955,153.358
C07254=1082.267,2.734,441.247,174.122,19.953,153.358
C07255=1082.262,2.484,441.261,174.120,19.950,153.358
C07256=1082.256,2.236,441.275,174.119,19.948,153.357
C07257=1082.251,1.986,441.289,174.117,19.946,153.357
C07258=1082.244,1.736,441.303,174.116,19.944,153.357
C07259=1082.238,1.486,441.317,174.114,19.942,153.357
C07260=1082.233,1.237,441.331,174.113,19.940,153.357
C07261=1082.227,0.988,441.345,174.111,19.938,153.357
C07262=1082.222,0.738,441.359,174.110,19.936,153.356
C07263=1082.215,0.488,441.373,174.108,19.933,153.356
C07264=1082.209,0.239,441.387,174.107,19.931,153.356
C07265=1082.204,-0.011,441.400,174.106,19.929,153.356
C07266=1082.198,-0.260,441.414,174.104,19.927,153.356
C07267=1082.193,-0.510,441.428,174.103,19.925,153.355
C07268=1082.186,-0.786,441.443,174.101,19.923,153.355
C07269=1082.180,-1.062,441.459,174.100,19.921,153.355
C07270=1082.173,-1.337,441.474,174.098,19.918,153.355
C07271=1082.167,-1.613,441.490,174.097,19.915,153.355
C07272=1082.161,-1.862,441.503,174.094,19.913,153.355
C07273=1082.155,-2.112,441.517,174.093,19.911,153.354
C07274=1082.150,-2.361,441.531,174.092,19.909,153.354
C07275=1082.144,-2.611,441.546,174.091,19.907,153.354
C07276=1082.138,-2.861,441.560,174.089,19.904,153.354
C07277=1082.132,-3.110,441.573,174.087,19.902,153.354
C07278=1082.126,-3.359,441.587,174.086,19.900,153.354
C07279=1082.121,-3.609,441.601,174.085,19.898,153.353
C07280=1082.115,-3.858,441.614,174.083,19.896,153.353
C07281=1082.109,-4.108,441.628,174.081,19.894,153.353
C07282=1082.102,-4.358,441.641,174.080,19.892,153.353
C07283=1082.097,-4.607,441.655,174.079,19.890,153.353
